# B&R Automation Studio project NAEUL004C00R13L518F00 (part 23)

#### Act_OptP0939FBCtrl.st
```iecst
ACTION Act_OptP0939FBCtrl:

	fbJogSlowToFastDlyTm.PT	:= T#2s;
	fbJogSlowToFastDlyTm;
	fbLmtRstTm;

	//Lifter Safety Sensor Interruption
	IF EDGENEG(p_tyDI.bLifterSafetyLmtSW1 AND p_tyDI.bLifterSafetyLmtSW2 AND p_tyDI.bLifterTimingBeltSen) THEN
		tyP0939Lifter2.tyMotionStd.tyBtnStop.bRtCompl	:= TRUE;
	END_IF

//	IF EDGEPOS((p_udiLifter2AxisErrID = 21570 OR p_udiLifter2AxisErrID = 21571)
	IF EDGEPOS((p_bLifter2FwdLmtSen OR p_bLifter2RevLmtSen OR p_udiLifter2AxisErrID = 21570 OR p_udiLifter2AxisErrID = 21571)
		AND tyP0939Lifter2.tyMotionStd.tyBtnJogDown.bValue = FALSE
		AND tyP0939Lifter2.tyMotionStd.tyBtnJogUp.bValue = FALSE)
	THEN
		fbLmtRstTm.IN				:= TRUE;
	END_IF

	IF fbLmtRstTm.Q = TRUE THEN
		tyP0939Lifter2.tyMotionStd.tyBtnRst.bRtCompl		:= TRUE;
	END_IF

	IF (tyP0939Lifter2.tyMotionStd.tyBtnJogUp.bValue = FALSE AND tyP0939Lifter2.tyMotionStd.tyBtnJogDown.bValue = FALSE) AND (p_bLifter2Jogging = TRUE) THEN
		bJogStopLifter	:= TRUE;
	END_IF

	IF tyP0939Lifter2.tyMotionStd.tyBtnStop.bRtCompl = TRUE THEN
		eLifter2Act		:= LifterActStop;

		IF p_eLifter2Stat = LifterActStop AND p_eLifter2Status = Done THEN
			eLifter2Act	:= LifterActIdle;

			tyP0939Lifter2.tyMotionStd.tyBtnStop.bRtCompl			:= FALSE;
			tyP0939Lifter2.tyMotionStd.tyBtnJogDown.bRtCompl			:= FALSE;
			tyP0939Lifter2.tyMotionStd.tyBtnJogUp.bRtCompl			:= FALSE;
			tyP0939Lifter2.tyMotionStd.tyBtnOrigin.bRtCompl			:= FALSE;
			tyP0939Lifter2.tyMotionStd.tyBtnMovAbs.bRtCompl			:= FALSE;
			tyP0939Lifter2.tyMotionStd.tyBtnMovRel.bRtCompl			:= FALSE;
			tyP0939Lifter2.tyLifter.tyBtnGo.bRtCompl				:= FALSE;
			tyP0939Lifter2.tyLifter.tyBtnNxtSlt.bRtCompl			:= FALSE;
			tyP0939Lifter2.tyLifter.tyBtnPrevSlt.bRtCompl			:= FALSE;
			tyP0939Lifter2.tyLifter.tyBtnGoLaneA.bRtCompl			:= FALSE;
			tyP0939Lifter2.tyLifter.tyBtnGoLaneB.bRtCompl			:= FALSE;
			tyP0939Lifter2.tyLifter.tyBtnGoLaneD_G.bRtCompl			:= FALSE;
			tyP0939Lifter2.tyLifter.tyBtnGoLaneE_H.bRtCompl			:= FALSE;

			tyP0939Lifter2.tyMotionStd.tyBtnStop.bValue				:= TRUE;
			tyP0939Lifter2.tyMotionStd.tyBtnJogDown.bValue			:= FALSE;
			tyP0939Lifter2.tyMotionStd.tyBtnJogUp.bValue				:= FALSE;
			tyP0939Lifter2.tyMotionStd.tyBtnOrigin.bValue			:= FALSE;
			tyP0939Lifter2.tyMotionStd.tyBtnMovAbs.bValue			:= FALSE;
			tyP0939Lifter2.tyMotionStd.tyBtnMovRel.bValue			:= FALSE;
			tyP0939Lifter2.tyLifter.tyBtnGo.bValue					:= FALSE;
			tyP0939Lifter2.tyLifter.tyBtnNxtSlt.bValue				:= FALSE;
			tyP0939Lifter2.tyLifter.tyBtnPrevSlt.bValue				:= FALSE;
			tyP0939Lifter2.tyLifter.tyBtnGoLaneA.bValue				:= FALSE;
			tyP0939Lifter2.tyLifter.tyBtnGoLaneB.bValue				:= FALSE;
			tyP0939Lifter2.tyLifter.tyBtnGoLaneD_G.bValue			:= FALSE;
			tyP0939Lifter2.tyLifter.tyBtnGoLaneE_H.bValue			:= FALSE;

			tyP0939Lifter2.tyMotionStd.tyBtnStop.bRtLk				:= TRUE;
			tyP0939Lifter2.tyMotionStd.tyBtnJogDown.bRtLk			:= FALSE;
			tyP0939Lifter2.tyMotionStd.tyBtnJogUp.bRtLk				:= FALSE;
			tyP0939Lifter2.tyMotionStd.tyBtnOrigin.bRtLk				:= FALSE;
			tyP0939Lifter2.tyMotionStd.tyBtnMovAbs.bRtLk				:= FALSE;
			tyP0939Lifter2.tyMotionStd.tyBtnMovRel.bRtLk				:= FALSE;
			tyP0939Lifter2.tyLifter.tyBtnGo.bRtLk					:= FALSE;
			tyP0939Lifter2.tyLifter.tyBtnNxtSlt.bRtLk				:= FALSE;
			tyP0939Lifter2.tyLifter.tyBtnPrevSlt.bRtLk				:= FALSE;
			tyP0939Lifter2.tyLifter.tyBtnGoLaneA.bRtLk				:= FALSE;
			tyP0939Lifter2.tyLifter.tyBtnGoLaneB.bRtLk				:= FALSE;
			tyP0939Lifter2.tyLifter.tyBtnGoLaneD_G.bRtLk			:= FALSE;
			tyP0939Lifter2.tyLifter.tyBtnGoLaneE_H.bRtLk			:= FALSE;

		END_IF

	ELSIF (tyP0939Lifter2.tyMotionStd.tyBtnJogDown.bRtCompl = TRUE) OR (tyP0939Lifter2.tyMotionStd.tyBtnJogUp.bRtCompl = TRUE) OR (bJogStopLifter = TRUE) THEN
		bJogSlow					:= FALSE;
		bJogFast					:= FALSE;
		fbJogSlowToFastDlyTm.IN		:= FALSE;

		eLifter2Act		:= LifterActJogStop;

		IF p_eLifter2Stat = LifterActJogStop AND p_eLifter2Status = Done THEN
			eLifter2Act		:= LifterActIdle;

			bJogStopLifter	:= FALSE;

			tyP0939Lifter2.tyMotionStd.tyBtnStop.bRtCompl			:= FALSE;
			tyP0939Lifter2.tyMotionStd.tyBtnJogDown.bRtCompl		:= FALSE;
			tyP0939Lifter2.tyMotionStd.tyBtnJogUp.bRtCompl			:= FALSE;
			tyP0939Lifter2.tyMotionStd.tyBtnOrigin.bRtCompl			:= FALSE;
			tyP0939Lifter2.tyMotionStd.tyBtnMovAbs.bRtCompl			:= FALSE;
			tyP0939Lifter2.tyMotionStd.tyBtnMovRel.bRtCompl			:= FALSE;
			tyP0939Lifter2.tyLifter.tyBtnGo.bRtCompl				:= FALSE;
			tyP0939Lifter2.tyLifter.tyBtnNxtSlt.bRtCompl			:= FALSE;
			tyP0939Lifter2.tyLifter.tyBtnPrevSlt.bRtCompl			:= FALSE;
			tyP0939Lifter2.tyLifter.tyBtnGoLaneA.bRtCompl			:= FALSE;
			tyP0939Lifter2.tyLifter.tyBtnGoLaneB.bRtCompl			:= FALSE;
			tyP0939Lifter2.tyLifter.tyBtnGoLaneD_G.bRtCompl			:= FALSE;
			tyP0939Lifter2.tyLifter.tyBtnGoLaneE_H.bRtCompl			:= FALSE;

			tyP0939Lifter2.tyMotionStd.tyBtnStop.bValue				:= TRUE;
			tyP0939Lifter2.tyMotionStd.tyBtnJogDown.bValue			:= FALSE;
			tyP0939Lifter2.tyMotionStd.tyBtnJogUp.bValue			:= FALSE;
			tyP0939Lifter2.tyMotionStd.tyBtnOrigin.bValue			:= FALSE;
			tyP0939Lifter2.tyMotionStd.tyBtnMovAbs.bValue			:= FALSE;
			tyP0939Lifter2.tyMotionStd.tyBtnMovRel.bValue			:= FALSE;
			tyP0939Lifter2.tyLifter.tyBtnGo.bValue					:= FALSE;
			tyP0939Lifter2.tyLifter.tyBtnNxtSlt.bValue				:= FALSE;
			tyP0939Lifter2.tyLifter.tyBtnPrevSlt.bValue				:= FALSE;
			tyP0939Lifter2.tyLifter.tyBtnGoLaneA.bValue				:= FALSE;
			tyP0939Lifter2.tyLifter.tyBtnGoLaneB.bValue				:= FALSE;
			tyP0939Lifter2.tyLifter.tyBtnGoLaneD_G.bValue			:= FALSE;
			tyP0939Lifter2.tyLifter.tyBtnGoLaneE_H.bValue			:= FALSE;

			tyP0939Lifter2.tyMotionStd.tyBtnStop.bRtLk				:= TRUE;
			tyP0939Lifter2.tyMotionStd.tyBtnJogDown.bRtLk			:= FALSE;
			tyP0939Lifter2.tyMotionStd.tyBtnJogUp.bRtLk				:= FALSE;
			tyP0939Lifter2.tyMotionStd.tyBtnOrigin.bRtLk			:= FALSE;
			tyP0939Lifter2.tyMotionStd.tyBtnMovAbs.bRtLk			:= FALSE;
			tyP0939Lifter2.tyMotionStd.tyBtnMovRel.bRtLk			:= FALSE;
			tyP0939Lifter2.tyLifter.tyBtnGo.bRtLk					:= FALSE;
			tyP0939Lifter2.tyLifter.tyBtnNxtSlt.bRtLk				:= FALSE;
			tyP0939Lifter2.tyLifter.tyBtnPrevSlt.bRtLk				:= FALSE;
			tyP0939Lifter2.tyLifter.tyBtnGoLaneA.bRtLk				:= FALSE;
			tyP0939Lifter2.tyLifter.tyBtnGoLaneB.bRtLk				:= FALSE;
			tyP0939Lifter2.tyLifter.tyBtnGoLaneD_G.bRtLk			:= FALSE;
			tyP0939Lifter2.tyLifter.tyBtnGoLaneE_H.bRtLk			:= FALSE;

		END_IF

	ELSIF tyP0939Lifter2.tyMotionStd.tyBtnPwr.bRtCompl = TRUE THEN
		tyP0939Lifter2.tyMotionStd.tyBtnPwr.bRtLk					:= TRUE;

		IF tyP0939Lifter2.tyMotionStd.tyBtnPwr.bValue = TRUE THEN
			eLifter2Act		:= LifterActPwrOn;

			IF p_eLifter2Stat = LifterActPwrOn AND p_eLifter2Status = Done THEN
				eLifter2Act	:= LifterActIdle;

				tyP0939Lifter2.tyMotionStd.tyBtnPwr.bRtCompl		:= FALSE;
				tyP0939Lifter2.tyMotionStd.tyBtnPwr.bRtLk		:= FALSE;
			END_IF
		ELSE
			eLifter2Act		:= LifterActPwrOff;

			IF p_eLifter2Stat = LifterActPwrOff AND p_eLifter2Status = Done THEN
				eLifter2Act	:= LifterActIdle;

				tyP0939Lifter2.tyMotionStd.tyBtnPwr.bRtCompl		:= FALSE;
				tyP0939Lifter2.tyMotionStd.tyBtnPwr.bRtLk		:= FALSE;
			END_IF
		END_IF

	ELSIF tyP0939Lifter2.tyMotionStd.tyBtnOrigin.bRtCompl = TRUE THEN
		tyP0939Lifter2.tyMotionStd.tyBtnOrigin.bValue				:= TRUE;
		tyP0939Lifter2.tyMotionStd.tyBtnStop.bValue					:= FALSE;

		tyP0939Lifter2.tyMotionStd.tyBtnOrigin.bRtLk					:= TRUE;
		tyP0939Lifter2.tyMotionStd.tyBtnStop.bRtLk					:= FALSE;

		eLifter2Act		:= LifterActHoming;

		IF p_eLifter2Stat = LifterActHoming AND p_eLifter2Status = Done THEN
			eLifter2Act	:= LifterActIdle;

			tyP0939Lifter2.tyMotionStd.tyBtnOrigin.bRtCompl		:= FALSE;
			tyP0939Lifter2.tyMotionStd.tyBtnOrigin.bValue		:= FALSE;
			tyP0939Lifter2.tyMotionStd.tyBtnStop.bValue			:= TRUE;

			tyP0939Lifter2.tyMotionStd.tyBtnOrigin.bRtLk			:= FALSE;
			tyP0939Lifter2.tyMotionStd.tyBtnStop.bRtLk			:= TRUE;

		END_IF

	ELSIF tyP0939Lifter2.tyMotionStd.tyBtnRst.bRtCompl = TRUE THEN
		tyP0939Lifter2.tyMotionStd.tyBtnRst.bValue				:= TRUE;
		tyP0939Lifter2.tyMotionStd.tyBtnRst.bRtLk				:= TRUE;

		eLifter2Act		:= LifterActRstAxisErr;

		IF p_eLifter2Stat = LifterActRstAxisErr AND p_eLifter2Status = Done THEN
			eLifter2Act	:= LifterActIdle;

			tyP0939Lifter2.tyMotionStd.tyBtnRst.bRtCompl			:= FALSE;
			tyP0939Lifter2.tyMotionStd.tyBtnRst.bValue			:= FALSE;
			tyP0939Lifter2.tyMotionStd.tyBtnRst.bRtLk			:= FALSE;

			fbLmtRstTm.IN			:= FALSE;
		END_IF

	ELSIF tyP0939Lifter2.tyLifter.tyBtnGo.bRtCompl = TRUE THEN
		tyP0939Lifter2.tyLifter.tyBtnGo.bValue				:= TRUE;
		tyP0939Lifter2.tyMotionStd.tyBtnStop.bValue			:= FALSE;

		tyP0939Lifter2.tyLifter.tyBtnGo.bRtLk				:= TRUE;
		tyP0939Lifter2.tyMotionStd.tyBtnStop.bRtLk			:= FALSE;

		(*diMnlLifterMag1GoSlt2	:= tyP0939Lifter2.tyLifter.tyNumNewSlt.diValue;*)
		diMnlLifterNomSpd2		:= tyP0939Lifter2.tyMotionStd.tyNumNomSpd.diValue;

		CASE tyP0939Lifter2.tyLifter.tyNumMagPos.diValue OF
			1:
				eLifter2Act	:= LifterActGoASltPos;
				diMnlLifterMag1GoSlt2	:= tyP0939Lifter2.tyLifter.tyNumNewSlt.diValue;

			2:
				eLifter2Act	:= LifterActGoBSltPos;
				diMnlLifterMag2GoSlt2	:= tyP0939Lifter2.tyLifter.tyNumNewSlt.diValue;

			3:
				eLifter2Act	:= LifterActGoCSltPos;
				diMnlLifterMag3GoSlt2	:= tyP0939Lifter2.tyLifter.tyNumNewSlt.diValue;

			4:
				eLifter2Act	:= LifterActGoDSltPos;
				diMnlLifterMag3GoSlt2	:= tyP0939Lifter2.tyLifter.tyNumNewSlt.diValue;
		END_CASE

		IF (p_eLifter2Stat = LifterActGoASltPos
			OR p_eLifter2Stat = LifterActGoBSltPos
			OR p_eLifter2Stat = LifterActGoCSltPos
			OR p_eLifter2Stat = LifterActGoDSltPos)
			AND p_eLifter2Status = Done THEN
			eLifter2Act	:= LifterActIdle;

			tyP0939Lifter2.tyLifter.tyBtnGo.bRtCompl				:= FALSE;
			tyP0939Lifter2.tyLifter.tyBtnGo.bValue				:= FALSE;
			tyP0939Lifter2.tyMotionStd.tyBtnStop.bValue			:= TRUE;

			tyP0939Lifter2.tyLifter.tyBtnGo.bRtLk				:= FALSE;
			tyP0939Lifter2.tyMotionStd.tyBtnStop.bRtLk			:= TRUE;
		END_IF

	ELSIF tyP0939Lifter2.tyLifter.tyBtnNxtSlt.bRtCompl = TRUE THEN
		tyP0939Lifter2.tyLifter.tyBtnNxtSlt.bValue				:= TRUE;
		tyP0939Lifter2.tyMotionStd.tyBtnStop.bValue				:= FALSE;

		tyP0939Lifter2.tyLifter.tyBtnNxtSlt.bRtLk				:= TRUE;
		tyP0939Lifter2.tyMotionStd.tyBtnStop.bRtLk				:= FALSE;

		(*diMnlLifterMag1GoSlt2	:= tyP0939Lifter2.tyLifter.tyNumNewSlt.diValue;*)
		diMnlLifterNomSpd2		:= tyP0939Lifter2.tyMotionStd.tyNumNomSpd.diValue;

		CASE tyP0939Lifter2.tyLifter.tyNumMagPos.diValue OF
			1:
				eLifter2Act	:= LifterActGoNxtASltPos;
				diMnlLifterMag1GoSlt2	:= tyP0939Lifter2.tyLifter.tyNumNewSlt.diValue;
			2:
				eLifter2Act	:= LifterActGoNxtBSltPos;
				diMnlLifterMag2GoSlt2	:= tyP0939Lifter2.tyLifter.tyNumNewSlt.diValue;
			3:
				eLifter2Act	:= LifterActGoNxtCSltPos;
				diMnlLifterMag3GoSlt2	:= tyP0939Lifter2.tyLifter.tyNumNewSlt.diValue;
			4:
				eLifter2Act	:= LifterActGoNxtDSltPos;
		//		diMnlLifterMag4GoSlt	:= tyP0939Lifter2.tyLifter.tyNumNewSlt.diValue;

		END_CASE

		IF (p_eLifter2Stat = LifterActGoNxtASltPos
			OR p_eLifter2Stat = LifterActGoNxtBSltPos
			OR p_eLifter2Stat = LifterActGoNxtCSltPos
			OR p_eLifter2Stat = LifterActGoNxtDSltPos)
			AND p_eLifter2Status = Done THEN
			eLifter2Act	:= LifterActIdle;

			tyP0939Lifter2.tyLifter.tyBtnNxtSlt.bRtCompl				:= FALSE;
			tyP0939Lifter2.tyLifter.tyBtnNxtSlt.bValue				:= FALSE;
			tyP0939Lifter2.tyMotionStd.tyBtnStop.bValue				:= TRUE;

			tyP0939Lifter2.tyLifter.tyBtnNxtSlt.bRtLk				:= FALSE;
			tyP0939Lifter2.tyMotionStd.tyBtnStop.bRtLk				:= TRUE;
		END_IF

	ELSIF tyP0939Lifter2.tyLifter.tyBtnPrevSlt.bRtCompl = TRUE THEN
		tyP0939Lifter2.tyLifter.tyBtnPrevSlt.bValue				:= TRUE;
		tyP0939Lifter2.tyMotionStd.tyBtnStop.bValue				:= FALSE;

		tyP0939Lifter2.tyLifter.tyBtnPrevSlt.bRtLk				:= TRUE;
		tyP0939Lifter2.tyMotionStd.tyBtnStop.bRtLk				:= FALSE;

	//	diMnlLifterMag1GoSlt2	:= tyP0939Lifter2.tyLifter.tyNumNewSlt.diValue;
		diMnlLifterNomSpd2		:= tyP0939Lifter2.tyMotionStd.tyNumNomSpd.diValue;

		CASE tyP0939Lifter2.tyLifter.tyNumMagPos.diValue OF

			1:
				eLifter2Act	:= LifterActGoPrevASltPos;
				diMnlLifterMag1GoSlt2	:= tyP0939Lifter2.tyLifter.tyNumNewSlt.diValue;

			2:
				eLifter2Act	:= LifterActGoPrevBSltPos;
				diMnlLifterMag2GoSlt2	:= tyP0939Lifter2.tyLifter.tyNumNewSlt.diValue;

			3:
				eLifter2Act	:= LifterActGoPrevCSltPos;
				diMnlLifterMag3GoSlt2	:= tyP0939Lifter2.tyLifter.tyNumNewSlt.diValue;

			4:
				eLifter2Act	:= LifterActGoPrevDSltPos;
		//		diMnlLifterMag4GoSlt	:= tyP0939Lifter2.tyLifter.tyNumNewSlt.diValue;

		END_CASE

		IF (p_eLifter2Stat = LifterActGoPrevASltPos
			OR p_eLifter2Stat = LifterActGoPrevBSltPos
			OR p_eLifter2Stat = LifterActGoPrevCSltPos
			OR p_eLifter2Stat = LifterActGoPrevDSltPos)
			AND p_eLifter2Status = Done THEN
			eLifter2Act	:= LifterActIdle;

			tyP0939Lifter2.tyLifter.tyBtnPrevSlt.bRtCompl				:= FALSE;
			tyP0939Lifter2.tyLifter.tyBtnPrevSlt.bValue					:= FALSE;
			tyP0939Lifter2.tyMotionStd.tyBtnStop.bValue					:= TRUE;

			tyP0939Lifter2.tyLifter.tyBtnPrevSlt.bRtLk					:= FALSE;
			tyP0939Lifter2.tyMotionStd.tyBtnStop.bRtLk					:= TRUE;
		END_IF

	ELSIF tyP0939Lifter2.tyLifter.tyBtnGoLaneA.bRtCompl = TRUE THEN
		tyP0939Lifter2.tyLifter.tyBtnGoLaneA.bValue	:= TRUE;
		tyP0939Lifter2.tyMotionStd.tyBtnStop.bValue	:= FALSE;

		tyP0939Lifter2.tyLifter.tyBtnGoLaneA.bRtLk	:= TRUE;
		tyP0939Lifter2.tyMotionStd.tyBtnStop.bRtLk	:= FALSE;

		diMnlLifterNomSpd2	:= tyP0939Lifter2.tyMotionStd.tyNumNomSpd.diValue;

		eLifter2Act	:= LifterActGoAPos;

		IF p_eLifter2Stat = LifterActGoAPos AND p_eLifter2Status = Done THEN
			eLifter2Act	:= LifterActIdle;

			tyP0939Lifter2.tyLifter.tyBtnGoLaneA.bRtCompl	:= FALSE;

			tyP0939Lifter2.tyLifter.tyBtnGoLaneA.bValue	:= FALSE;
			tyP0939Lifter2.tyMotionStd.tyBtnStop.bValue	:= TRUE;

			tyP0939Lifter2.tyLifter.tyBtnGoLaneA.bRtLk	:= FALSE;
			tyP0939Lifter2.tyMotionStd.tyBtnStop.bRtLk	:= TRUE;
		END_IF

	ELSIF tyP0939Lifter2.tyLifter.tyBtnGoLaneB.bRtCompl = TRUE THEN
		tyP0939Lifter2.tyLifter.tyBtnGoLaneB.bValue	:= TRUE;
		tyP0939Lifter2.tyMotionStd.tyBtnStop.bValue	:= FALSE;

		tyP0939Lifter2.tyLifter.tyBtnGoLaneB.bRtLk	:= TRUE;
		tyP0939Lifter2.tyMotionStd.tyBtnStop.bRtLk	:= FALSE;

		diMnlLifterNomSpd2	:= tyP0939Lifter2.tyMotionStd.tyNumNomSpd.diValue;

		eLifter2Act	:= LifterActGoBPos;

		IF p_eLifter2Stat = LifterActGoBPos AND p_eLifter2Status = Done THEN
			eLifter2Act	:= LifterActIdle;

			tyP0939Lifter2.tyLifter.tyBtnGoLaneB.bRtCompl	:= FALSE;

			tyP0939Lifter2.tyLifter.tyBtnGoLaneB.bValue	:= FALSE;
			tyP0939Lifter2.tyMotionStd.tyBtnStop.bValue	:= TRUE;

			tyP0939Lifter2.tyLifter.tyBtnGoLaneB.bRtLk	:= FALSE;
			tyP0939Lifter2.tyMotionStd.tyBtnStop.bRtLk	:= TRUE;
		END_IF

	ELSIF tyP0939Lifter2.tyLifter.tyBtnGoLaneD_G.bRtCompl = TRUE THEN
		tyP0939Lifter2.tyLifter.tyBtnGoLaneD_G.bValue	:= TRUE;
		tyP0939Lifter2.tyMotionStd.tyBtnStop.bValue	:= FALSE;

		tyP0939Lifter2.tyLifter.tyBtnGoLaneD_G.bRtLk	:= TRUE;
		tyP0939Lifter2.tyMotionStd.tyBtnStop.bRtLk	:= FALSE;

		diMnlLifterNomSpd2	:= tyP0939Lifter2.tyMotionStd.tyNumNomSpd.diValue;

		eLifter2Act	:= LifterActGoGPos;

		IF p_eLifter2Stat = LifterActGoGPos AND p_eLifter2Status = Done THEN
			eLifter2Act	:= LifterActIdle;

			tyP0939Lifter2.tyLifter.tyBtnGoLaneD_G.bRtCompl	:= FALSE;

			tyP0939Lifter2.tyLifter.tyBtnGoLaneD_G.bValue	:= FALSE;
			tyP0939Lifter2.tyMotionStd.tyBtnStop.bValue	:= TRUE;

			tyP0939Lifter2.tyLifter.tyBtnGoLaneD_G.bRtLk	:= FALSE;
			tyP0939Lifter2.tyMotionStd.tyBtnStop.bRtLk	:= TRUE;
		END_IF

	ELSIF tyP0939Lifter2.tyLifter.tyBtnGoLaneE_H.bRtCompl = TRUE THEN
		tyP0939Lifter2.tyLifter.tyBtnGoLaneE_H.bValue	:= TRUE;
		tyP0939Lifter2.tyMotionStd.tyBtnStop.bValue	:= FALSE;

		tyP0939Lifter2.tyLifter.tyBtnGoLaneE_H.bRtLk	:= TRUE;
		tyP0939Lifter2.tyMotionStd.tyBtnStop.bRtLk	:= FALSE;

		diMnlLifterNomSpd2	:= tyP0939Lifter2.tyMotionStd.tyNumNomSpd.diValue;

		eLifter2Act	:= LifterActGoHPos;

		IF p_eLifter2Stat = LifterActGoHPos AND p_eLifter2Status = Done THEN
			eLifter2Act	:= LifterActIdle;

			tyP0939Lifter2.tyLifter.tyBtnGoLaneE_H.bRtCompl	:= FALSE;

			tyP0939Lifter2.tyLifter.tyBtnGoLaneE_H.bValue	:= FALSE;
			tyP0939Lifter2.tyMotionStd.tyBtnStop.bValue	:= TRUE;

			tyP0939Lifter2.tyLifter.tyBtnGoLaneE_H.bRtLk	:= FALSE;
			tyP0939Lifter2.tyMotionStd.tyBtnStop.bRtLk	:= TRUE;
		END_IF
	ELSIF tyP0939Lifter2.tyMotionStd.tyBtnMovAbs.bRtCompl = TRUE THEN

		tyP0939Lifter2.tyMotionStd.tyBtnMovAbs.bValue				:= TRUE;
		tyP0939Lifter2.tyMotionStd.tyBtnStop.bValue					:= FALSE;

		tyP0939Lifter2.tyMotionStd.tyBtnMovAbs.bRtLk					:= TRUE;
		tyP0939Lifter2.tyMotionStd.tyBtnStop.bRtLk					:= FALSE;

		diMnlLifterTargetPos2	:= tyP0939Lifter2.tyMotionStd.tyNumTargetPos.diValue;
		diMnlLifterNomSpd2		:= tyP0939Lifter2.tyMotionStd.tyNumNomSpd.diValue;

		eLifter2Act			:= LifterActMovAbs;

		IF p_eLifter2Stat = LifterActMovAbs AND p_eLifter2Status = Done THEN
			eLifter2Act	:= LifterActIdle;

			tyP0939Lifter2.tyMotionStd.tyBtnMovAbs.bRtCompl		:= FALSE;
			tyP0939Lifter2.tyMotionStd.tyBtnMovAbs.bValue		:= FALSE;
			tyP0939Lifter2.tyMotionStd.tyBtnStop.bValue			:= TRUE;

			tyP0939Lifter2.tyMotionStd.tyBtnMovAbs.bRtLk			:= FALSE;
			tyP0939Lifter2.tyMotionStd.tyBtnStop.bRtLk			:= TRUE;
		END_IF

	ELSIF tyP0939Lifter2.tyMotionStd.tyBtnMovRel.bRtCompl = TRUE THEN
		tyP0939Lifter2.tyMotionStd.tyBtnMovRel.bValue			:= TRUE;
		tyP0939Lifter2.tyMotionStd.tyBtnStop.bValue				:= FALSE;

		tyP0939Lifter2.tyMotionStd.tyBtnMovRel.bRtLk				:= TRUE;
		tyP0939Lifter2.tyMotionStd.tyBtnStop.bRtLk				:= FALSE;

		diMnlLifterStepSize2		:= tyP0939Lifter2.tyMotionStd.tyNumStepSize.diValue;
		diMnlLifterNomSpd2		:= tyP0939Lifter2.tyMotionStd.tyNumNomSpd.diValue;

		eLifter2Act		:= LifterActMovRel;

		IF p_eLifter2Stat = LifterActMovRel AND p_eLifter2Status = Done THEN
			eLifter2Act	:= LifterActIdle;

			tyP0939Lifter2.tyMotionStd.tyBtnMovRel.bRtCompl		:= FALSE;
			tyP0939Lifter2.tyMotionStd.tyBtnMovRel.bValue		:= FALSE;
			tyP0939Lifter2.tyMotionStd.tyBtnStop.bValue			:= TRUE;

			tyP0939Lifter2.tyMotionStd.tyBtnMovRel.bRtLk			:= FALSE;
			tyP0939Lifter2.tyMotionStd.tyBtnStop.bRtLk			:= TRUE;

		END_IF

	ELSIF (tyP0939Lifter2.tyMotionStd.tyBtnJogDown.bValue = TRUE) AND (fbJogSlowToFastDlyTm.Q = FALSE) AND (bJogSlow = FALSE) THEN
		tyP0939Lifter2.tyMotionStd.tyBtnStop.bValue				:= FALSE;
		tyP0939Lifter2.tyMotionStd.tyBtnStop.bRtLk				:= FALSE;

		fbJogSlowToFastDlyTm.IN		:= TRUE;

		diMnlLifterJogSpd2	:= tyP0939Lifter2.tyMotionStd.tyNumSlwSpd.diValue;

		eLifter2Act		:= LifterActJogDown;

		IF p_eLifter2Stat = LifterActJogDown AND p_eLifter2Status = Done THEN

			eLifter2Act	:= LifterActIdle;
			bJogSlow				:= TRUE;

		ELSIF p_eLifter2Status = Error THEN

			fbJogSlowToFastDlyTm.IN	:= FALSE;
			bJogSlow				:= TRUE;

		END_IF

	ELSIF (tyP0939Lifter2.tyMotionStd.tyBtnJogDown.bValue = TRUE) AND (fbJogSlowToFastDlyTm.Q = TRUE) AND (bJogFast = FALSE) THEN
		tyP0939Lifter2.tyMotionStd.tyBtnStop.bValue					:= FALSE;
		tyP0939Lifter2.tyMotionStd.tyBtnStop.bRtLk					:= FALSE;

		fbJogSlowToFastDlyTm.IN		:= TRUE;

		diMnlLifterJogSpd2	:= tyP0939Lifter2.tyMotionStd.tyNumNomSpd.diValue;

		eLifter2Act		:= LifterActJogDown;

		IF p_eLifter2Stat = LifterActJogDown AND p_eLifter2Status = Done THEN
			eLifter2Act	:= LifterActIdle;
			bJogFast				:= TRUE;
		ELSIF p_eLifter2Status = Error THEN
			fbJogSlowToFastDlyTm.IN	:= FALSE;
			bJogFast				:= TRUE;
		END_IF

	ELSIF (tyP0939Lifter2.tyMotionStd.tyBtnJogUp.bValue = TRUE) AND (fbJogSlowToFastDlyTm.Q = FALSE) AND (bJogSlow = FALSE) THEN
		tyP0939Lifter2.tyMotionStd.tyBtnStop.bValue				:= FALSE;
		tyP0939Lifter2.tyMotionStd.tyBtnStop.bRtLk				:= FALSE;

		fbJogSlowToFastDlyTm.IN		:= TRUE;

		diMnlLifterJogSpd2	:= tyP0939Lifter2.tyMotionStd.tyNumSlwSpd.diValue;

		eLifter2Act		:= LifterActJogUp;

		IF p_eLifter2Stat = LifterActJogUp AND p_eLifter2Status = Done THEN
			eLifter2Act	:= LifterActIdle;
			bJogSlow				:= TRUE;

		ELSIF p_eLifter2Status = Error THEN
			fbJogSlowToFastDlyTm.IN	:= FALSE;
			bJogSlow				:= TRUE;
		END_IF

	ELSIF (tyP0939Lifter2.tyMotionStd.tyBtnJogUp.bValue = TRUE) AND (fbJogSlowToFastDlyTm.Q = TRUE) AND (bJogFast = FALSE) THEN

		tyP0939Lifter2.tyMotionStd.tyBtnStop.bValue				:= FALSE;
		tyP0939Lifter2.tyMotionStd.tyBtnStop.bRtLk				:= FALSE;

		fbJogSlowToFastDlyTm.IN		:= TRUE;

		diMnlLifterJogSpd2	:= tyP0939Lifter2.tyMotionStd.tyNumNomSpd.diValue;

		eLifter2Act		:= LifterActJogUp;

		IF p_eLifter2Stat = LifterActJogUp AND p_eLifter2Status = Done THEN
			eLifter2Act	:= LifterActIdle;
			bJogFast	:= TRUE;

		ELSIF p_eLifter2Status = Error THEN
			fbJogSlowToFastDlyTm.IN	:= FALSE;
			bJogFast				:= TRUE;
		END_IF
	END_IF

	//Shutter Control
	IF tyP0939Lifter2.tyInOutletShutterFB.tyBtnOpen.bRtCompl = TRUE THEN
		tyP0939Lifter2.tyInOutletShutterFB.tyBtnOpen.bRtCompl	:= FALSE;

		tyP0939Lifter2.tyInOutletShutterFB.tyBtnOpen.bValue	:= TRUE;
		tyP0939Lifter2.tyInOutletShutterFB.tyBtnClose.bValue	:= FALSE;

	ELSIF tyP0939Lifter2.tyInOutletShutterFB.tyBtnClose.bRtCompl = TRUE THEN
		tyP0939Lifter2.tyInOutletShutterFB.tyBtnClose.bRtCompl	:= FALSE;

		tyP0939Lifter2.tyInOutletShutterFB.tyBtnClose.bValue	:= TRUE;
		tyP0939Lifter2.tyInOutletShutterFB.tyBtnOpen.bValue	:= FALSE;
	END_IF

	IF tyP0939Lifter2.tyInOutletShutterFB.tyBtnOpen.bValue = TRUE THEN
		eInShutterAct	:= PneuActRet;
		eOutShutterAct	:= PneuActRet;

		IF (p_eInShutterStat = PneuActRet AND p_eInShutterStatus = Done)
			AND (p_eOutShutterStat = PneuActRet AND p_eOutShutterStatus = Done)
			THEN
			eInShutterAct	:= PneuActIdle;
			eOutShutterAct	:= PneuActIdle;
			tyP0939Lifter2.tyInOutletShutterFB.tyBtnOpen.bValue	:= FALSE;
		ELSIF p_eInShutterStatus = Error OR p_eOutShutterStatus = Error THEN
			tyP0939Lifter2.tyInOutletShutterFB.tyBtnOpen.bValue	:= FALSE;
		END_IF

	ELSIF tyP0939Lifter2.tyInOutletShutterFB.tyBtnClose.bValue = TRUE THEN
		eInShutterAct	:= PneuActExt;
		eOutShutterAct	:= PneuActExt;
		IF (p_eInShutterStat = PneuActExt AND p_eInShutterStatus = Done)
			AND (p_eOutShutterStat = PneuActExt AND p_eOutShutterStatus = Done)
			THEN
			eInShutterAct	:= PneuActIdle;
			eOutShutterAct	:= PneuActIdle;
			tyP0939Lifter2.tyInOutletShutterFB.tyBtnClose.bValue := FALSE;
		ELSIF p_eInShutterStatus = Error OR p_eOutShutterStatus = Error THEN
			tyP0939Lifter2.tyInOutletShutterFB.tyBtnClose.bValue := FALSE;
		END_IF
	END_IF

END_ACTION
```

#### Act_OptP0939FBStat.st
```iecst
ACTION Act_OptP0939FBStat:

	IF p_bLifter2AxisErr = TRUE THEN
		tyP0939Lifter2.tyMotionStd.tyStringStat.sValue	:= p_sLifter2AxisErrTxt;
	ELSE
		IF NOT(p_bLifter2Jogging AND p_eLifter2Stat = LifterActIdle) THEN
			tyP0939Lifter2.tyMotionStd.tyStringStat.sValue	:= p_sLifter2StatTxt;
		END_IF
	END_IF

END_ACTION
```

#### Act_OptP0939Mask.st
```iecst
ACTION Act_OptP0939Mask:

	// Interlock Power
	IF p_bLifter2AxisErr = TRUE AND p_bLifter2PwrOn = FALSE THEN
		fUIInRtStatOff(ADR(tyP0939Lifter2.tyMotionStd.tyBtnPwr.uiMaskRtStat));
		tyP0939Lifter2.tyMotionStd.tyBtnPwr.bValue		:= FALSE;
	ELSE
		fUIInRtStatHide(ADR(tyP0939Lifter2.tyMotionStd.tyBtnPwr.uiMaskRtStat));
	END_IF

	// Interlock Others Move
	IF p_bLifter2AxisErr = TRUE OR p_bLifter2PwrOn = FALSE THEN
		fUIInRtStatOff(ADR(tyP0939Lifter2.tyMotionStd.tyBtnOrigin.uiMaskRtStat));
		fUIInRtStatOff(ADR(tyP0939Lifter2.tyMotionStd.tyBtnMovRel.uiMaskRtStat));
		fUIInRtStatOff(ADR(tyP0939Lifter2.tyMotionStd.tyBtnJogUp.uiMaskRtStat));
		fUIInRtStatOff(ADR(tyP0939Lifter2.tyMotionStd.tyBtnJogDown.uiMaskRtStat));
	ELSE
		fUIInRtStatHide(ADR(tyP0939Lifter2.tyMotionStd.tyBtnOrigin.uiMaskRtStat));
		fUIInRtStatHide(ADR(tyP0939Lifter2.tyMotionStd.tyBtnMovRel.uiMaskRtStat));
		fUIInRtStatHide(ADR(tyP0939Lifter2.tyMotionStd.tyBtnJogUp.uiMaskRtStat));
		fUIInRtStatHide(ADR(tyP0939Lifter2.tyMotionStd.tyBtnJogDown.uiMaskRtStat));
	END_IF

	// Interlock Move Absolute
	IF p_bLifter2AxisErr = TRUE OR p_bLifter2PwrOn = FALSE OR p_bLifter2IsHomed = FALSE THEN

		fUIInRtStatOff(ADR(tyP0939Lifter2.tyMotionStd.tyBtnMovAbs.uiMaskRtStat));

		fUIInRtStatOff(ADR(tyP0939Lifter2.tyLifter.tyBtnGo.uiMaskRtStat));
		fUIInRtStatOff(ADR(tyP0939Lifter2.tyLifter.tyBtnNxtSlt.uiMaskRtStat));
		fUIInRtStatOff(ADR(tyP0939Lifter2.tyLifter.tyBtnPrevSlt.uiMaskRtStat));
		fUIInRtStatOff(ADR(tyP0939Lifter2.tyLifter.tyBtnGoLaneA.uiMaskRtStat));
		fUIInRtStatOff(ADR(tyP0939Lifter2.tyLifter.tyBtnGoLaneB.uiMaskRtStat));
		fUIInRtStatOff(ADR(tyP0939Lifter2.tyLifter.tyBtnGoLaneD_G.uiMaskRtStat));
		fUIInRtStatOff(ADR(tyP0939Lifter2.tyLifter.tyBtnGoLaneE_H.uiMaskRtStat));

	ELSE
		fUIInRtStatHide(ADR(tyP0939Lifter2.tyMotionStd.tyBtnMovAbs.uiMaskRtStat));

		fUIInRtStatHide(ADR(tyP0939Lifter2.tyLifter.tyBtnGo.uiMaskRtStat));
		fUIInRtStatHide(ADR(tyP0939Lifter2.tyLifter.tyBtnNxtSlt.uiMaskRtStat));
		fUIInRtStatHide(ADR(tyP0939Lifter2.tyLifter.tyBtnPrevSlt.uiMaskRtStat));
		fUIInRtStatHide(ADR(tyP0939Lifter2.tyLifter.tyBtnGoLaneA.uiMaskRtStat));
		fUIInRtStatHide(ADR(tyP0939Lifter2.tyLifter.tyBtnGoLaneB.uiMaskRtStat));
		fUIInRtStatHide(ADR(tyP0939Lifter2.tyLifter.tyBtnGoLaneD_G.uiMaskRtStat));
		fUIInRtStatHide(ADR(tyP0939Lifter2.tyLifter.tyBtnGoLaneE_H.uiMaskRtStat));

	END_IF

	//Interlock Limit Sensor
	IF tyP0939Lifter2.tyMotionStd.tyBtnDownLmtSen.bValue = TRUE THEN
		fUIInRtStatOff(ADR(tyP0939Lifter2.tyMotionStd.tyBtnJogDown.uiMaskRtStat));
	END_IF

	IF tyP0939Lifter2.tyMotionStd.tyBtnUpLmtSen.bValue = TRUE THEN
		fUIInRtStatOff(ADR(tyP0939Lifter2.tyMotionStd.tyBtnJogUp.uiMaskRtStat));
	END_IF

	// Interlock When Moving
	IF tyP0939Lifter2.tyMotionStd.tyBtnOrigin.bRtCompl = TRUE THEN

		fUIInRtStatOff(ADR(tyP0939Lifter2.tyMotionStd.tyBtnMovAbs.uiMaskRtStat));
		fUIInRtStatOff(ADR(tyP0939Lifter2.tyMotionStd.tyBtnMovRel.uiMaskRtStat));
		fUIInRtStatOff(ADR(tyP0939Lifter2.tyMotionStd.tyBtnJogUp.uiMaskRtStat));
		fUIInRtStatOff(ADR(tyP0939Lifter2.tyMotionStd.tyBtnJogDown.uiMaskRtStat));

		fUIInRtStatOff(ADR(tyP0939Lifter2.tyLifter.tyBtnGo.uiMaskRtStat));
		fUIInRtStatOff(ADR(tyP0939Lifter2.tyLifter.tyBtnPrevSlt.uiMaskRtStat));
		fUIInRtStatOff(ADR(tyP0939Lifter2.tyLifter.tyBtnNxtSlt.uiMaskRtStat));
		fUIInRtStatOff(ADR(tyP0939Lifter2.tyLifter.tyBtnGoLaneA.uiMaskRtStat));
		fUIInRtStatOff(ADR(tyP0939Lifter2.tyLifter.tyBtnGoLaneB.uiMaskRtStat));
		fUIInRtStatOff(ADR(tyP0939Lifter2.tyLifter.tyBtnGoLaneD_G.uiMaskRtStat));
		fUIInRtStatOff(ADR(tyP0939Lifter2.tyLifter.tyBtnGoLaneE_H.uiMaskRtStat));

	ELSIF tyP0939Lifter2.tyMotionStd.tyBtnMovAbs.bRtCompl = TRUE THEN

		fUIInRtStatOff(ADR(tyP0939Lifter2.tyMotionStd.tyBtnOrigin.uiMaskRtStat));
		fUIInRtStatOff(ADR(tyP0939Lifter2.tyMotionStd.tyBtnMovRel.uiMaskRtStat));
		fUIInRtStatOff(ADR(tyP0939Lifter2.tyMotionStd.tyBtnJogUp.uiMaskRtStat));
		fUIInRtStatOff(ADR(tyP0939Lifter2.tyMotionStd.tyBtnJogDown.uiMaskRtStat));

		fUIInRtStatOff(ADR(tyP0939Lifter2.tyLifter.tyBtnGo.uiMaskRtStat));
		fUIInRtStatOff(ADR(tyP0939Lifter2.tyLifter.tyBtnPrevSlt.uiMaskRtStat));
		fUIInRtStatOff(ADR(tyP0939Lifter2.tyLifter.tyBtnNxtSlt.uiMaskRtStat));
		fUIInRtStatOff(ADR(tyP0939Lifter2.tyLifter.tyBtnGoLaneA.uiMaskRtStat));
		fUIInRtStatOff(ADR(tyP0939Lifter2.tyLifter.tyBtnGoLaneB.uiMaskRtStat));
		fUIInRtStatOff(ADR(tyP0939Lifter2.tyLifter.tyBtnGoLaneD_G.uiMaskRtStat));
		fUIInRtStatOff(ADR(tyP0939Lifter2.tyLifter.tyBtnGoLaneE_H.uiMaskRtStat));

	ELSIF tyP0939Lifter2.tyMotionStd.tyBtnMovRel.bRtCompl = TRUE THEN

		fUIInRtStatOff(ADR(tyP0939Lifter2.tyMotionStd.tyBtnOrigin.uiMaskRtStat));
		fUIInRtStatOff(ADR(tyP0939Lifter2.tyMotionStd.tyBtnMovAbs.uiMaskRtStat));
		fUIInRtStatOff(ADR(tyP0939Lifter2.tyMotionStd.tyBtnJogUp.uiMaskRtStat));
		fUIInRtStatOff(ADR(tyP0939Lifter2.tyMotionStd.tyBtnJogDown.uiMaskRtStat));

		fUIInRtStatOff(ADR(tyP0939Lifter2.tyLifter.tyBtnGo.uiMaskRtStat));
		fUIInRtStatOff(ADR(tyP0939Lifter2.tyLifter.tyBtnNxtSlt.uiMaskRtStat));
		fUIInRtStatOff(ADR(tyP0939Lifter2.tyLifter.tyBtnPrevSlt.uiMaskRtStat));
		fUIInRtStatOff(ADR(tyP0939Lifter2.tyLifter.tyBtnGoLaneA.uiMaskRtStat));
		fUIInRtStatOff(ADR(tyP0939Lifter2.tyLifter.tyBtnGoLaneB.uiMaskRtStat));
		fUIInRtStatOff(ADR(tyP0939Lifter2.tyLifter.tyBtnGoLaneD_G.uiMaskRtStat));
		fUIInRtStatOff(ADR(tyP0939Lifter2.tyLifter.tyBtnGoLaneE_H.uiMaskRtStat));

	ELSIF tyP0939Lifter2.tyMotionStd.tyBtnJogDown.bRtCompl = TRUE OR tyP0939Lifter2.tyMotionStd.tyBtnJogDown.bValue = TRUE THEN
		fUIInRtStatOff(ADR(tyP0939Lifter2.tyMotionStd.tyBtnOrigin.uiMaskRtStat));
		fUIInRtStatOff(ADR(tyP0939Lifter2.tyMotionStd.tyBtnMovAbs.uiMaskRtStat));
		fUIInRtStatOff(ADR(tyP0939Lifter2.tyMotionStd.tyBtnMovRel.uiMaskRtStat));
		fUIInRtStatOff(ADR(tyP0939Lifter2.tyMotionStd.tyBtnJogUp.uiMaskRtStat));

		fUIInRtStatOff(ADR(tyP0939Lifter2.tyLifter.tyBtnGo.uiMaskRtStat));
		fUIInRtStatOff(ADR(tyP0939Lifter2.tyLifter.tyBtnNxtSlt.uiMaskRtStat));
		fUIInRtStatOff(ADR(tyP0939Lifter2.tyLifter.tyBtnPrevSlt.uiMaskRtStat));
		fUIInRtStatOff(ADR(tyP0939Lifter2.tyLifter.tyBtnGoLaneA.uiMaskRtStat));
		fUIInRtStatOff(ADR(tyP0939Lifter2.tyLifter.tyBtnGoLaneB.uiMaskRtStat));
		fUIInRtStatOff(ADR(tyP0939Lifter2.tyLifter.tyBtnGoLaneD_G.uiMaskRtStat));
		fUIInRtStatOff(ADR(tyP0939Lifter2.tyLifter.tyBtnGoLaneE_H.uiMaskRtStat));

	ELSIF tyP0939Lifter2.tyMotionStd.tyBtnJogUp.bRtCompl = TRUE OR tyP0939Lifter2.tyMotionStd.tyBtnJogUp.bValue = TRUE THEN
		fUIInRtStatOff(ADR(tyP0939Lifter2.tyMotionStd.tyBtnOrigin.uiMaskRtStat));
		fUIInRtStatOff(ADR(tyP0939Lifter2.tyMotionStd.tyBtnMovAbs.uiMaskRtStat));
		fUIInRtStatOff(ADR(tyP0939Lifter2.tyMotionStd.tyBtnMovRel.uiMaskRtStat));
		fUIInRtStatOff(ADR(tyP0939Lifter2.tyMotionStd.tyBtnJogDown.uiMaskRtStat));

		fUIInRtStatOff(ADR(tyP0939Lifter2.tyLifter.tyBtnGo.uiMaskRtStat));
		fUIInRtStatOff(ADR(tyP0939Lifter2.tyLifter.tyBtnNxtSlt.uiMaskRtStat));
		fUIInRtStatOff(ADR(tyP0939Lifter2.tyLifter.tyBtnPrevSlt.uiMaskRtStat));
		fUIInRtStatOff(ADR(tyP0939Lifter2.tyLifter.tyBtnGoLaneA.uiMaskRtStat));
		fUIInRtStatOff(ADR(tyP0939Lifter2.tyLifter.tyBtnGoLaneB.uiMaskRtStat));
		fUIInRtStatOff(ADR(tyP0939Lifter2.tyLifter.tyBtnGoLaneD_G.uiMaskRtStat));
		fUIInRtStatOff(ADR(tyP0939Lifter2.tyLifter.tyBtnGoLaneE_H.uiMaskRtStat));

	ELSIF tyP0939Lifter2.tyLifter.tyBtnGo.bRtCompl = TRUE THEN
		fUIInRtStatOff(ADR(tyP0939Lifter2.tyMotionStd.tyBtnOrigin.uiMaskRtStat));
		fUIInRtStatOff(ADR(tyP0939Lifter2.tyMotionStd.tyBtnMovAbs.uiMaskRtStat));
		fUIInRtStatOff(ADR(tyP0939Lifter2.tyMotionStd.tyBtnMovRel.uiMaskRtStat));
		fUIInRtStatOff(ADR(tyP0939Lifter2.tyMotionStd.tyBtnJogUp.uiMaskRtStat));
		fUIInRtStatOff(ADR(tyP0939Lifter2.tyMotionStd.tyBtnJogDown.uiMaskRtStat));

		fUIInRtStatOff(ADR(tyP0939Lifter2.tyLifter.tyBtnNxtSlt.uiMaskRtStat));
		fUIInRtStatOff(ADR(tyP0939Lifter2.tyLifter.tyBtnPrevSlt.uiMaskRtStat));
		fUIInRtStatOff(ADR(tyP0939Lifter2.tyLifter.tyBtnGoLaneA.uiMaskRtStat));
		fUIInRtStatOff(ADR(tyP0939Lifter2.tyLifter.tyBtnGoLaneB.uiMaskRtStat));
		fUIInRtStatOff(ADR(tyP0939Lifter2.tyLifter.tyBtnGoLaneD_G.uiMaskRtStat));
		fUIInRtStatOff(ADR(tyP0939Lifter2.tyLifter.tyBtnGoLaneE_H.uiMaskRtStat));

	ELSIF tyP0939Lifter2.tyLifter.tyBtnNxtSlt.bRtCompl = TRUE THEN
		fUIInRtStatOff(ADR(tyP0939Lifter2.tyMotionStd.tyBtnOrigin.uiMaskRtStat));
		fUIInRtStatOff(ADR(tyP0939Lifter2.tyMotionStd.tyBtnMovAbs.uiMaskRtStat));
		fUIInRtStatOff(ADR(tyP0939Lifter2.tyMotionStd.tyBtnMovRel.uiMaskRtStat));
		fUIInRtStatOff(ADR(tyP0939Lifter2.tyMotionStd.tyBtnJogUp.uiMaskRtStat));
		fUIInRtStatOff(ADR(tyP0939Lifter2.tyMotionStd.tyBtnJogDown.uiMaskRtStat));

		fUIInRtStatOff(ADR(tyP0939Lifter2.tyLifter.tyBtnGo.uiMaskRtStat));
		fUIInRtStatOff(ADR(tyP0939Lifter2.tyLifter.tyBtnPrevSlt.uiMaskRtStat));
		fUIInRtStatOff(ADR(tyP0939Lifter2.tyLifter.tyBtnGoLaneA.uiMaskRtStat));
		fUIInRtStatOff(ADR(tyP0939Lifter2.tyLifter.tyBtnGoLaneB.uiMaskRtStat));
		fUIInRtStatOff(ADR(tyP0939Lifter2.tyLifter.tyBtnGoLaneD_G.uiMaskRtStat));
		fUIInRtStatOff(ADR(tyP0939Lifter2.tyLifter.tyBtnGoLaneE_H.uiMaskRtStat));

	ELSIF tyP0939Lifter2.tyLifter.tyBtnPrevSlt.bRtCompl = TRUE THEN
		fUIInRtStatOff(ADR(tyP0939Lifter2.tyMotionStd.tyBtnOrigin.uiMaskRtStat));
		fUIInRtStatOff(ADR(tyP0939Lifter2.tyMotionStd.tyBtnMovAbs.uiMaskRtStat));
		fUIInRtStatOff(ADR(tyP0939Lifter2.tyMotionStd.tyBtnMovRel.uiMaskRtStat));
		fUIInRtStatOff(ADR(tyP0939Lifter2.tyMotionStd.tyBtnJogUp.uiMaskRtStat));
		fUIInRtStatOff(ADR(tyP0939Lifter2.tyMotionStd.tyBtnJogDown.uiMaskRtStat));

		fUIInRtStatOff(ADR(tyP0939Lifter2.tyLifter.tyBtnGo.uiMaskRtStat));
		fUIInRtStatOff(ADR(tyP0939Lifter2.tyLifter.tyBtnNxtSlt.uiMaskRtStat));
		fUIInRtStatOff(ADR(tyP0939Lifter2.tyLifter.tyBtnGoLaneA.uiMaskRtStat));
		fUIInRtStatOff(ADR(tyP0939Lifter2.tyLifter.tyBtnGoLaneB.uiMaskRtStat));
		fUIInRtStatOff(ADR(tyP0939Lifter2.tyLifter.tyBtnGoLaneD_G.uiMaskRtStat));
		fUIInRtStatOff(ADR(tyP0939Lifter2.tyLifter.tyBtnGoLaneE_H.uiMaskRtStat));

	ELSIF tyP0939Lifter2.tyLifter.tyBtnGoLaneA.bRtCompl = TRUE THEN
		fUIInRtStatOff(ADR(tyP0939Lifter2.tyMotionStd.tyBtnOrigin.uiMaskRtStat));
		fUIInRtStatOff(ADR(tyP0939Lifter2.tyMotionStd.tyBtnMovAbs.uiMaskRtStat));
		fUIInRtStatOff(ADR(tyP0939Lifter2.tyMotionStd.tyBtnMovRel.uiMaskRtStat));
		fUIInRtStatOff(ADR(tyP0939Lifter2.tyMotionStd.tyBtnJogUp.uiMaskRtStat));
		fUIInRtStatOff(ADR(tyP0939Lifter2.tyMotionStd.tyBtnJogDown.uiMaskRtStat));

		fUIInRtStatOff(ADR(tyP0939Lifter2.tyLifter.tyBtnGo.uiMaskRtStat));
		fUIInRtStatOff(ADR(tyP0939Lifter2.tyLifter.tyBtnNxtSlt.uiMaskRtStat));
		fUIInRtStatOff(ADR(tyP0939Lifter2.tyLifter.tyBtnPrevSlt.uiMaskRtStat));
		fUIInRtStatOff(ADR(tyP0939Lifter2.tyLifter.tyBtnGoLaneB.uiMaskRtStat));
		fUIInRtStatOff(ADR(tyP0939Lifter2.tyLifter.tyBtnGoLaneE_H.uiMaskRtStat));

	ELSIF tyP0939Lifter2.tyLifter.tyBtnGoLaneB.bRtCompl = TRUE THEN
		fUIInRtStatOff(ADR(tyP0939Lifter2.tyMotionStd.tyBtnOrigin.uiMaskRtStat));
		fUIInRtStatOff(ADR(tyP0939Lifter2.tyMotionStd.tyBtnMovAbs.uiMaskRtStat));
		fUIInRtStatOff(ADR(tyP0939Lifter2.tyMotionStd.tyBtnMovRel.uiMaskRtStat));
		fUIInRtStatOff(ADR(tyP0939Lifter2.tyMotionStd.tyBtnJogUp.uiMaskRtStat));
		fUIInRtStatOff(ADR(tyP0939Lifter2.tyMotionStd.tyBtnJogDown.uiMaskRtStat));

		fUIInRtStatOff(ADR(tyP0939Lifter2.tyLifter.tyBtnGo.uiMaskRtStat));
		fUIInRtStatOff(ADR(tyP0939Lifter2.tyLifter.tyBtnNxtSlt.uiMaskRtStat));
		fUIInRtStatOff(ADR(tyP0939Lifter2.tyLifter.tyBtnPrevSlt.uiMaskRtStat));
		fUIInRtStatOff(ADR(tyP0939Lifter2.tyLifter.tyBtnGoLaneA.uiMaskRtStat));
		fUIInRtStatOff(ADR(tyP0939Lifter2.tyLifter.tyBtnGoLaneD_G.uiMaskRtStat));

	END_IF

	//Axis Error
	IF tyP0939Lifter2.tyMotionStd.tyBtnPwr.bRtCompl = TRUE THEN
		fUIInRtStatOff(ADR(tyP0939Lifter2.tyMotionStd.tyBtnRst.uiMaskRtStat));
	ELSE
		fUIInRtStatHide(ADR(tyP0939Lifter2.tyMotionStd.tyBtnRst.uiMaskRtStat));
	END_IF

	//Next Slot
	IF p_diLifter2CurrSltA >= p_tyProdRcpCurrRcp0.diMaxSltValue THEN
		fUIInRtStatOff(ADR(tyP0939Lifter2.tyLifter.tyBtnNxtSlt.uiMaskRtStat));
	END_IF

	//Previous Slot
	IF p_diLifter2CurrSltA <= p_tyProdRcpCurrRcp0.diMinSltValue THEN
		fUIInRtStatOff(ADR(tyP0939Lifter2.tyLifter.tyBtnPrevSlt.uiMaskRtStat));
	END_IF

END_ACTION
```

#### Act_OptP0939UpdtDat.st
```iecst
ACTION Act_OptP0939UpdtDat:

	tyP0939Lifter2.tyMotionStd.tyNumCurrPos.diValue			:= p_diLifter2ActualPos;
	tyP0939Lifter2.tyMotionStd.tyNumErrCode.diValue			:= UDINT_TO_DINT(p_udiLifter2AxisErrID);
	tyP0939Lifter2.tyMotionStd.tyBitmapPwr.usiValueIdx		:= BOOL_TO_USINT(p_bLifter2PwrOn);
	tyP0939Lifter2.tyMotionStd.tyBitmapRst.usiValueIdx		:= BOOL_TO_USINT(NOT p_bLifter2AxisErr);
	tyP0939Lifter2.tyMotionStd.tyBitmapOrigin.usiValueIdx	:= BOOL_TO_USINT(p_bLifter2IsHomed);
	tyP0939Lifter2.tyMotionStd.tyBtnUpLmtSen.bValue			:= p_bLifter2UpSen;
	tyP0939Lifter2.tyMotionStd.tyBtnDownLmtSen.bValue		:= p_bLifter2DownSen;

	//Machine Bitmap
	IF p_bLifter2IsHomed = TRUE THEN
		IF p_diLifter2ActualPos <= (p_tyNtParamCurr.tyUILifterTargetPos.diMax / 3) THEN
			tyP0939Lifter2.tyMotionStd.tyBitmapMc.uiValueIdx 	:= 2;
		ELSIF p_diLifter2ActualPos <= (p_tyNtParamCurr.tyUILifterTargetPos.diMax / 3 * 2) THEN
			tyP0939Lifter2.tyMotionStd.tyBitmapMc.uiValueIdx 	:= 3;
		ELSE
			tyP0939Lifter2.tyMotionStd.tyBitmapMc.uiValueIdx 	:= 4;
		END_IF
	ELSE
		tyP0939Lifter2.tyMotionStd.tyBitmapMc.uiValueIdx	:= 2;
	END_IF

//	IF p_tyNtParamCurr.eProjMag = ULMagTriple THEN
//		tyP0939Lifter2.tyMotionStd.tyBitmapMc.uiValueIdx	:= tyP0939Lifter2.tyMotionStd.tyBitmapMc.uiValueIdx + 100;
//	END_IF

	IF p_tyNtParamCurr.eProjMag = ULMagDual THEN
		IF p_tyNtParamCurr.bProjLifterMagPlatform AND p_tyNtParamCurr.bUIConvDirRL THEN
			IF 	tyP0939Lifter2.tyMotionStd.tyBitmapMc.uiValueIdx < 700 THEN
				tyP0939Lifter2.tyMotionStd.tyBitmapMc.uiValueIdx	:= tyP0939Lifter2.tyMotionStd.tyBitmapMc.uiValueIdx + 700;
			END_IF
		ELSIF p_tyNtParamCurr.bProjLifterMagPlatform THEN
			IF p_tyNtParamCurr.bProjMagConvLane2Prep = FALSE THEN
				IF 	tyP0939Lifter2.tyMotionStd.tyBitmapMc.uiValueIdx < 600 THEN
					tyP0939Lifter2.tyMotionStd.tyBitmapMc.uiValueIdx	:= tyP0939Lifter2.tyMotionStd.tyBitmapMc.uiValueIdx + 600;
				END_IF
			ELSE
				IF 	tyP0939Lifter2.tyMotionStd.tyBitmapMc.uiValueIdx < 903 THEN //Lifter 2 - 905,906,907
					tyP0939Lifter2.tyMotionStd.tyBitmapMc.uiValueIdx	:= tyP0939Lifter2.tyMotionStd.tyBitmapMc.uiValueIdx + 903;
				END_IF
			END_IF
		ELSIF p_tyNtParamCurr.bMagAutoVerifyPrep = FALSE THEN
			IF 	tyP0939Lifter2.tyMotionStd.tyBitmapMc.uiValueIdx < 100 THEN
				tyP0939Lifter2.tyMotionStd.tyBitmapMc.uiValueIdx	:= tyP0939Lifter2.tyMotionStd.tyBitmapMc.uiValueIdx + 300;
			END_IF
		ELSE
			IF 	tyP0939Lifter2.tyMotionStd.tyBitmapMc.uiValueIdx < 300 THEN
				tyP0939Lifter2.tyMotionStd.tyBitmapMc.uiValueIdx	:= tyP0939Lifter2.tyMotionStd.tyBitmapMc.uiValueIdx + 300;
			END_IF
		END_IF
	ELSIF p_tyNtParamCurr.eProjMag = ULMagTriple THEN
		IF p_tyNtParamCurr.bProjLifterMagPlatform AND p_tyNtParamCurr.bUIConvDirRL THEN
			IF 	tyP0939Lifter2.tyMotionStd.tyBitmapMc.uiValueIdx < 800 THEN
				tyP0939Lifter2.tyMotionStd.tyBitmapMc.uiValueIdx	:= tyP0939Lifter2.tyMotionStd.tyBitmapMc.uiValueIdx + 800;
			END_IF
		ELSIF p_tyNtParamCurr.bProjLifterMagPlatform THEN
			IF tyP0939Lifter2.tyMotionStd.tyBitmapMc.uiValueIdx < 500 THEN
				tyP0939Lifter2.tyMotionStd.tyBitmapMc.uiValueIdx	:= tyP0939Lifter2.tyMotionStd.tyBitmapMc.uiValueIdx + 500;
			END_IF
		ELSIF p_tyNtParamCurr.bMagAutoVerifyPrep = TRUE AND p_tyNtParamCurr.bProjMotorizedPusherPrep = FALSE THEN
			IF 	tyP0939Lifter2.tyMotionStd.tyBitmapMc.uiValueIdx < 200 THEN
				tyP0939Lifter2.tyMotionStd.tyBitmapMc.uiValueIdx	:= tyP0939Lifter2.tyMotionStd.tyBitmapMc.uiValueIdx + 200;
			END_IF
		ELSIF  p_tyNtParamCurr.bMagAutoVerifyPrep = FALSE AND p_tyNtParamCurr.bProjMotorizedPusherPrep = TRUE THEN
			IF 	tyP0939Lifter2.tyMotionStd.tyBitmapMc.uiValueIdx < 400 THEN
				tyP0939Lifter2.tyMotionStd.tyBitmapMc.uiValueIdx	:= tyP0939Lifter2.tyMotionStd.tyBitmapMc.uiValueIdx + 400;
			END_IF
		END_IF
	END_IF

END_ACTION
```

#### Act_OptP0939Keypad.st
```iecst
ACTION Act_OptP0939Keypad:

	IF fUIOutRtStatTPIsOpen(ADR(tyP0939Lifter2.tyMotionStd.tyNumTargetPos.uiRtStat)) = TRUE THEN
		tyProperty.tyKeypad.tyStringTitle.sKeypadTitle	:= tyP0939Lifter2.tyMotionStd.tyNumTargetPos.sKeypadTitle;

	ELSIF fUIOutRtStatTPIsOpen(ADR(tyP0939Lifter2.tyMotionStd.tyNumStepSize.uiRtStat)) = TRUE THEN
		tyProperty.tyKeypad.tyStringTitle.sKeypadTitle	:= tyP0939Lifter2.tyMotionStd.tyNumStepSize.sKeypadTitle;

	ELSIF fUIOutRtStatTPIsOpen(ADR(tyP0939Lifter2.tyMotionStd.tyNumNomSpd.uiRtStat)) = TRUE THEN
		tyProperty.tyKeypad.tyStringTitle.sKeypadTitle	:= tyP0939Lifter2.tyMotionStd.tyNumNomSpd.sKeypadTitle;

	ELSIF fUIOutRtStatTPIsOpen(ADR(tyP0939Lifter2.tyMotionStd.tyNumSlwSpd.uiRtStat)) = TRUE THEN
		tyProperty.tyKeypad.tyStringTitle.sKeypadTitle	:= tyP0939Lifter2.tyMotionStd.tyNumSlwSpd.sKeypadTitle;

	ELSIF fUIOutRtStatTPIsOpen(ADR(tyP0939Lifter2.tyLifter.tyNumNewSlt.uiRtStat)) = TRUE THEN
		tyProperty.tyKeypad.tyStringTitle.sKeypadTitle	:= tyP0939Lifter2.tyLifter.tyNumNewSlt.sKeypadTitle;

	ELSIF fUIOutRtStatTPIsOpen(ADR(tyP0939Lifter2.tyLifter.tyNumMagPos.uiRtStat)) = TRUE THEN
		tyProperty.tyKeypad.tyStringTitle.sKeypadTitle	:= tyP0939Lifter2.tyLifter.tyNumMagPos.sKeypadTitle;

	END_IF

END_ACTION
```

#### Act_OptP0939RstMnl.st
```iecst
ACTION Act_OptP0939RstMnl:

	IF EDGEPOS((bManualMod = FALSE) OR (p_eLifter2Status = Error)) THEN

		eLifter2Act	:= LifterActIdle;

		bJogSlow				:= FALSE;
		bJogFast				:= FALSE;
		fbJogSlowToFastDlyTm.IN	:= FALSE;

		tyP0939Lifter2.tyLifter.tyBtnGo.bRtCompl					:= FALSE;
		tyP0939Lifter2.tyLifter.tyBtnNxtSlt.bRtCompl				:= FALSE;
		tyP0939Lifter2.tyLifter.tyBtnPrevSlt.bRtCompl			:= FALSE;
		tyP0939Lifter2.tyLifter.tyBtnGoLaneA.bRtCompl			:= FALSE;
		tyP0939Lifter2.tyLifter.tyBtnGoLaneB.bRtCompl			:= FALSE;
		tyP0939Lifter2.tyLifter.tyBtnGoLaneD_G.bRtCompl			:= FALSE;
		tyP0939Lifter2.tyLifter.tyBtnGoLaneE_H.bRtCompl			:= FALSE;

		tyP0939Lifter2.tyLifter.tyBtnGo.bValue					:= FALSE;
		tyP0939Lifter2.tyLifter.tyBtnNxtSlt.bValue				:= FALSE;
		tyP0939Lifter2.tyLifter.tyBtnPrevSlt.bValue				:= FALSE;
		tyP0939Lifter2.tyLifter.tyBtnGoLaneA.bValue				:= FALSE;
		tyP0939Lifter2.tyLifter.tyBtnGoLaneB.bValue				:= FALSE;
		tyP0939Lifter2.tyLifter.tyBtnGoLaneD_G.bValue				:= FALSE;
		tyP0939Lifter2.tyLifter.tyBtnGoLaneE_H.bValue				:= FALSE;

		tyP0939Lifter2.tyLifter.tyBtnGo.bRtLk					:= FALSE;
		tyP0939Lifter2.tyLifter.tyBtnNxtSlt.bRtLk				:= FALSE;
		tyP0939Lifter2.tyLifter.tyBtnPrevSlt.bRtLk				:= FALSE;
		tyP0939Lifter2.tyLifter.tyBtnGoLaneA.bRtLk				:= FALSE;
		tyP0939Lifter2.tyLifter.tyBtnGoLaneB.bRtLk				:= FALSE;
		tyP0939Lifter2.tyLifter.tyBtnGoLaneD_G.bRtLk				:= FALSE;
		tyP0939Lifter2.tyLifter.tyBtnGoLaneE_H.bRtLk				:= FALSE;

		tyP0939Lifter2.tyLifter.tyBtnGo.uiMaskRtStat.0			:= FALSE;
		tyP0939Lifter2.tyLifter.tyBtnNxtSlt.uiMaskRtStat.0		:= FALSE;
		tyP0939Lifter2.tyLifter.tyBtnPrevSlt.uiMaskRtStat.0		:= FALSE;
		tyP0939Lifter2.tyLifter.tyBtnGoLaneA.uiMaskRtStat.0		:= FALSE;
		tyP0939Lifter2.tyLifter.tyBtnGoLaneB.uiMaskRtStat.0		:= FALSE;
		tyP0939Lifter2.tyLifter.tyBtnGoLaneD_G.uiMaskRtStat.0		:= FALSE;
		tyP0939Lifter2.tyLifter.tyBtnGoLaneE_H.uiMaskRtStat.0		:= FALSE;

		tyP0939Lifter2.tyMotionStd.tyBtnPwr.bRtCompl				:= FALSE;
		tyP0939Lifter2.tyMotionStd.tyBtnStop.bRtCompl			:= FALSE;
		tyP0939Lifter2.tyMotionStd.tyBtnOrigin.bRtCompl			:= FALSE;
		tyP0939Lifter2.tyMotionStd.tyBtnRst.bRtCompl				:= FALSE;
		tyP0939Lifter2.tyMotionStd.tyBtnMovAbs.bRtCompl			:= FALSE;
		tyP0939Lifter2.tyMotionStd.tyBtnMovRel.bRtCompl			:= FALSE;
		tyP0939Lifter2.tyMotionStd.tyBtnJogUp.bRtCompl			:= FALSE;
		tyP0939Lifter2.tyMotionStd.tyBtnJogDown.bRtCompl			:= FALSE;

		tyP0939Lifter2.tyMotionStd.tyBtnPwr.bValue				:= FALSE;
		tyP0939Lifter2.tyMotionStd.tyBtnStop.bValue				:= TRUE;
		tyP0939Lifter2.tyMotionStd.tyBtnOrigin.bValue			:= FALSE;
		tyP0939Lifter2.tyMotionStd.tyBtnRst.bValue				:= FALSE;
		tyP0939Lifter2.tyMotionStd.tyBtnMovAbs.bValue			:= FALSE;
		tyP0939Lifter2.tyMotionStd.tyBtnMovRel.bValue			:= FALSE;
		tyP0939Lifter2.tyMotionStd.tyBtnJogUp.bValue				:= FALSE;
		tyP0939Lifter2.tyMotionStd.tyBtnJogDown.bValue			:= FALSE;

		tyP0939Lifter2.tyMotionStd.tyBtnPwr.bRtLk				:= FALSE;
		tyP0939Lifter2.tyMotionStd.tyBtnStop.bRtLk				:= TRUE;
		tyP0939Lifter2.tyMotionStd.tyBtnOrigin.bRtLk				:= FALSE;
		tyP0939Lifter2.tyMotionStd.tyBtnRst.bRtLk				:= FALSE;
		tyP0939Lifter2.tyMotionStd.tyBtnMovAbs.bRtLk				:= FALSE;
		tyP0939Lifter2.tyMotionStd.tyBtnMovRel.bRtLk				:= FALSE;
		tyP0939Lifter2.tyMotionStd.tyBtnJogUp.bRtLk				:= FALSE;
		tyP0939Lifter2.tyMotionStd.tyBtnJogDown.bRtLk			:= FALSE;

		tyP0939Lifter2.tyMotionStd.tyBtnPwr.uiMaskRtStat			:= TRUE;
		tyP0939Lifter2.tyMotionStd.tyBtnOrigin.uiMaskRtStat		:= FALSE;
		tyP0939Lifter2.tyMotionStd.tyBtnRst.uiMaskRtStat			:= TRUE;
		tyP0939Lifter2.tyMotionStd.tyBtnMovAbs.uiMaskRtStat		:= FALSE;
		tyP0939Lifter2.tyMotionStd.tyBtnMovRel.uiMaskRtStat		:= FALSE;
		tyP0939Lifter2.tyMotionStd.tyBtnJogUp.uiMaskRtStat		:= FALSE;
		tyP0939Lifter2.tyMotionStd.tyBtnJogDown.uiMaskRtStat		:= FALSE;

	END_IF

	eInShutterAct	:= PneuActIdle;
	eOutShutterAct	:= PneuActIdle;

	tyP0939Lifter2.tyInOutletShutterFB.tyBtnClose.bRtCompl	:= FALSE;
	tyP0939Lifter2.tyInOutletShutterFB.tyBtnClose.bValue	:= FALSE;
	tyP0939Lifter2.tyInOutletShutterFB.tyBtnOpen.bRtCompl	:= FALSE;
	tyP0939Lifter2.tyInOutletShutterFB.tyBtnOpen.bValue	:= FALSE;

END_ACTION
```

#### Act_EntP0940Disp.st
```iecst
ACTION Act_EntP0940Disp:

	//Access Address
	p_tyC0005Main ACCESS ADR(tyCommon.tyMain);

	p_tyC0007Notif ACCESS ADR(tyCommon.tyNotif);

	p_tyC0008MsgBox ACCESS ADR(tyP0940CommCtrl.tyMsgBoxHide);

	p_tyC0009Info ACCESS ADR(tyCommon.tyInfo);

	p_tyP0940CommCtrlUSSMEMAA ACCESS ADR(tyP0940CommCtrl.tyUSSMEMAA);
	p_tyP0940CommCtrlUSSMEMAB ACCESS ADR(tyP0940CommCtrl.tyUSSMEMAB);
	p_tyP0940CommCtrlSOT ACCESS ADR(tyP0940CommCtrl.tySOT);
	p_tyP0940CommDMCRFID ACCESS ADR(tyP0940CommCtrl.tyDMCRFID);
	//Upstream Line A
	IF p_tyMcParamCurr.tyUSCommASMEMA.bStatSigSetGd = TRUE THEN
		tyP0940CommCtrl.tyUSSMEMAA.tyBtnUBAStat.usiTxtIdx	:= 0;
	ELSE
		tyP0940CommCtrl.tyUSSMEMAA.tyBtnUBAStat.usiTxtIdx	:= 1;
	END_IF

	tyP0940CommCtrl.tyUSSMEMAA.tyBtnUBAStat.uiRtStat.0	:= NOT(p_tyMcParamCurr.tyUSCommASMEMA.eSelection = SMEMASelIPC9851Ext);

	//Upstream Line B
	IF p_tyMcParamCurr.tyUSCommBSMEMA.bStatSigSetGd = TRUE THEN
		tyP0940CommCtrl.tyUSSMEMAB.tyBtnUBAStat.usiTxtIdx	:= 0;
	ELSE
		tyP0940CommCtrl.tyUSSMEMAB.tyBtnUBAStat.usiTxtIdx	:= 1;
	END_IF

	tyP0940CommCtrl.tyUSSMEMAB.tyBtnUBAStat.uiRtStat.0	:= NOT(p_tyMcParamCurr.tyUSCommBSMEMA.eSelection = SMEMASelIPC9851Ext);

	CASE p_tyMcParamCurr.eAGVComProtocol OF
		McSetAGVCommOPCUA:
			tyP0940CommCtrl.tySOT.tyTxtAIVCommProtocol.usiValueIdx := 0;

		McSetAGVCommHardIO:
			tyP0940CommCtrl.tySOT.tyTxtAIVCommProtocol.usiValueIdx := 1;

		McSetAGVCommDisabled:
			tyP0940CommCtrl.tySOT.tyTxtAIVCommProtocol.usiValueIdx := 2;

	END_CASE

END_ACTION
```

#### Act_OptP0940FullMask.st
```iecst
ACTION Act_OptP0940FullMask:

	IF eCurrPage = UIP0940CommCtrl THEN

		IF p_tyDI.bEStopSig = FALSE THEN
			p_tyC0002FullMask ACCESS ADR(tyP0940CommCtrl.tyFullMaskEStop);

		ELSIF p_tyDI.bCoverSWSig = FALSE THEN
			p_tyC0002FullMask ACCESS ADR(tyP0940CommCtrl.tyFullMaskCWSig);

		ELSIF p_tyDI.bSafetyRlySig = FALSE THEN
			p_tyC0002FullMask ACCESS ADR(tyP0940CommCtrl.tyFullMaskSafetyRly);

		ELSE
			p_tyC0002FullMask ACCESS ADR(tyP0940CommCtrl.tyFullMaskHide);

		END_IF

	END_IF

END_ACTION
```

#### Act_OptP0940ReadDI.st
```iecst
ACTION Act_OptP0940ReadDI:

		tyP0940CommCtrl.tyUSSMEMAA.tyBtnUBA.bValue		:= p_tyDI.bUBAA;
		tyP0940CommCtrl.tyUSSMEMAA.tyBtnUBAStat.bValue	:= p_tyDI.bUBAAStat;
		tyP0940CommCtrl.tyUSSMEMAB.tyBtnUBA.bValue		:= p_tyDI.bUBAB;
		tyP0940CommCtrl.tyUSSMEMAB.tyBtnUBAStat.bValue	:= p_tyDI.bUBABStat;

	IF p_tyNtParamCurr.bProjSOTSensorPrep THEN
//		CASE p_tyMcParamCurr.eAGVComProtocol OF
//			McSetAGVCommHardIO, :
				tyP0940CommCtrl.tySOT.tyBtnAIVRcv1.bValue		:= p_tyDI.bSOT1Receive;
				tyP0940CommCtrl.tySOT.tyBtnAIVErr1.bValue		:= p_tyDI.bSOT1AIVError;
				tyP0940CommCtrl.tySOT.tyBtnAIVRdy1.bValue		:= p_tyDI.bSOT1AIVReady;
				tyP0940CommCtrl.tySOT.tyBtnAIVAvail1.bValue		:= p_tyDI.bSOT1AIVAvailable;
				tyP0940CommCtrl.tySOT.tyBtnAIVSLarge1.bValue	:= p_tyDI.bSOT1AIVSizeLarge;

				tyP0940CommCtrl.tySOT.tyBtnAIVRcv2.bValue		:= p_tyDI.bSOT2Receive;
				tyP0940CommCtrl.tySOT.tyBtnAIVErr2.bValue		:= p_tyDI.bSOT2AIVError;
				tyP0940CommCtrl.tySOT.tyBtnAIVRdy2.bValue		:= p_tyDI.bSOT2AIVReady;
				tyP0940CommCtrl.tySOT.tyBtnAIVAvail2.bValue		:= p_tyDI.bSOT2AIVAvailable;
				tyP0940CommCtrl.tySOT.tyBtnAIVSLarge2.bValue	:= p_tyDI.bSOT2AIVSizeLarge;

				tyP0940CommCtrl.tySOT.tyBtnAIVRcv3.bValue		:= p_tyDI.bSOT3Receive;
				tyP0940CommCtrl.tySOT.tyBtnAIVErr3.bValue		:= p_tyDI.bSOT3AIVError;
				tyP0940CommCtrl.tySOT.tyBtnAIVRdy3.bValue		:= p_tyDI.bSOT3AIVReady;
				tyP0940CommCtrl.tySOT.tyBtnAIVAvail3.bValue		:= p_tyDI.bSOT3AIVAvailable;
				tyP0940CommCtrl.tySOT.tyBtnAIVSLarge3.bValue	:= p_tyDI.bSOT3AIVSizeLarge;

				tyP0940CommCtrl.tySOT.tyBtnAIVRcv4.bValue		:= p_tyDI.bSOT4Receive;
				tyP0940CommCtrl.tySOT.tyBtnAIVErr4.bValue		:= p_tyDI.bSOT4AIVError;
				tyP0940CommCtrl.tySOT.tyBtnAIVRdy4.bValue		:= p_tyDI.bSOT4AIVReady;
				tyP0940CommCtrl.tySOT.tyBtnAIVAvail4.bValue		:= p_tyDI.bSOT4AIVAvailable;
				tyP0940CommCtrl.tySOT.tyBtnAIVSLarge4.bValue	:= p_tyDI.bSOT4AIVSizeLarge;

				tyP0940CommCtrl.tySOT.tyBtnFleetMgrActive.bValue := p_tyDI.bFleetManagerReady OR p_tyTagFromMes.bActive;

//			McSetAGVCommOPCUA:
//
//				tyP0940CommCtrl.tySOT.tyBtnAIVErr1.bValue		:= p_tyTagFromMes.tyTagStatOfPlatforms[1].bError;
//				tyP0940CommCtrl.tySOT.tyBtnAIVRdy1.bValue		:= p_tyTagFromMes.tyTagStatOfPlatforms[1].bReady;
//				tyP0940CommCtrl.tySOT.tyBtnAIVAvail1.bValue		:= p_tyTagFromMes.tyTagStatOfPlatforms[1].bAvailable;
//				tyP0940CommCtrl.tySOT.tyBtnAIVSLarge1.bValue	:= p_tyTagFromMes.tyTagStatOfPlatforms[1].bSizeLarge;
//
//				tyP0940CommCtrl.tySOT.tyBtnAIVErr2.bValue		:= p_tyTagFromMes.tyTagStatOfPlatforms[2].bError;
//				tyP0940CommCtrl.tySOT.tyBtnAIVRdy2.bValue		:= p_tyTagFromMes.tyTagStatOfPlatforms[2].bReady;
//				tyP0940CommCtrl.tySOT.tyBtnAIVAvail2.bValue		:= p_tyTagFromMes.tyTagStatOfPlatforms[2].bAvailable;
//				tyP0940CommCtrl.tySOT.tyBtnAIVSLarge2.bValue	:= p_tyTagFromMes.tyTagStatOfPlatforms[2].bSizeLarge;
//
//				tyP0940CommCtrl.tySOT.tyBtnAIVErr3.bValue		:= p_tyTagFromMes.tyTagStatOfPlatforms[3].bError;
//				tyP0940CommCtrl.tySOT.tyBtnAIVRdy3.bValue		:= p_tyTagFromMes.tyTagStatOfPlatforms[3].bReady;
//				tyP0940CommCtrl.tySOT.tyBtnAIVAvail3.bValue		:= p_tyTagFromMes.tyTagStatOfPlatforms[3].bAvailable;
//				tyP0940CommCtrl.tySOT.tyBtnAIVSLarge3.bValue	:= p_tyTagFromMes.tyTagStatOfPlatforms[3].bSizeLarge;
//
//				tyP0940CommCtrl.tySOT.tyBtnAIVErr4.bValue		:= p_tyTagFromMes.tyTagStatOfPlatforms[4].bError;
//				tyP0940CommCtrl.tySOT.tyBtnAIVRdy4.bValue		:= p_tyTagFromMes.tyTagStatOfPlatforms[4].bReady;
//				tyP0940CommCtrl.tySOT.tyBtnAIVAvail4.bValue		:= p_tyTagFromMes.tyTagStatOfPlatforms[4].bAvailable;
//				tyP0940CommCtrl.tySOT.tyBtnAIVSLarge4.bValue	:= p_tyTagFromMes.tyTagStatOfPlatforms[4].bSizeLarge;
//
//				tyP0940CommCtrl.tySOT.tyBtnFleetMgrActive.bValue := p_tyTagFromMes.bActive;

//		END_CASE
	ELSIF p_tyMcParamCurr.eAGVComProtocol = McSetAGVCommHardIO AND p_tyNtParamCurr.bProjSOTSensorPrep = FALSE THEN
		tyP0940CommCtrl.tySOT.tyBtnAIVRcv1.bValue		:= p_tyDI.bSOT1Receive;
		tyP0940CommCtrl.tySOT.tyBtnAIVErr1.bValue		:= p_tyDI.bSOT1AIVError;
		tyP0940CommCtrl.tySOT.tyBtnAIVRdy1.bValue		:= p_tyDI.bSOT1AIVReady;
		tyP0940CommCtrl.tySOT.tyBtnAIVAvail1.bValue		:= p_tyDI.bSOT1AIVAvailable;
		tyP0940CommCtrl.tySOT.tyBtnAIVSLarge1.bValue	:= p_tyDI.bSOT1AIVSizeLarge;

		tyP0940CommCtrl.tySOT.tyBtnAIVRcv2.bValue		:= p_tyDI.bSOT2Receive;
		tyP0940CommCtrl.tySOT.tyBtnAIVErr2.bValue		:= p_tyDI.bSOT2AIVError;
		tyP0940CommCtrl.tySOT.tyBtnAIVRdy2.bValue		:= p_tyDI.bSOT2AIVReady;
		tyP0940CommCtrl.tySOT.tyBtnAIVAvail2.bValue		:= p_tyDI.bSOT2AIVAvailable;
		tyP0940CommCtrl.tySOT.tyBtnAIVSLarge2.bValue	:= p_tyDI.bSOT2AIVSizeLarge;

		tyP0940CommCtrl.tySOT.tyBtnAIVRcv3.bValue		:= p_tyDI.bSOT3Receive;
		tyP0940CommCtrl.tySOT.tyBtnAIVErr3.bValue		:= p_tyDI.bSOT3AIVError;
		tyP0940CommCtrl.tySOT.tyBtnAIVRdy3.bValue		:= p_tyDI.bSOT3AIVReady;
		tyP0940CommCtrl.tySOT.tyBtnAIVAvail3.bValue		:= p_tyDI.bSOT3AIVAvailable;
		tyP0940CommCtrl.tySOT.tyBtnAIVSLarge3.bValue	:= p_tyDI.bSOT3AIVSizeLarge;

		tyP0940CommCtrl.tySOT.tyBtnAIVRcv4.bValue		:= p_tyDI.bSOT4Receive;
		tyP0940CommCtrl.tySOT.tyBtnAIVErr4.bValue		:= p_tyDI.bSOT4AIVError;
		tyP0940CommCtrl.tySOT.tyBtnAIVRdy4.bValue		:= p_tyDI.bSOT4AIVReady;
		tyP0940CommCtrl.tySOT.tyBtnAIVAvail4.bValue		:= p_tyDI.bSOT4AIVAvailable;
		tyP0940CommCtrl.tySOT.tyBtnAIVSLarge4.bValue	:= p_tyDI.bSOT4AIVSizeLarge;

		tyP0940CommCtrl.tySOT.tyBtnFleetMgrActive.bValue := p_tyDI.bFleetManagerReady;

	ELSIF p_tyMcParamCurr.eAGVComProtocol = McSetAGVCommOPCUA AND p_tyNtParamCurr.bProjSOTSensorPrep = FALSE THEN

		tyP0940CommCtrl.tySOT.tyBtnAIVErr1.bValue		:= p_tyTagFromMes.tyTagStatOfPlatforms[1].bError;
		tyP0940CommCtrl.tySOT.tyBtnAIVRdy1.bValue		:= p_tyTagFromMes.tyTagStatOfPlatforms[1].bReady;
		tyP0940CommCtrl.tySOT.tyBtnAIVAvail1.bValue		:= p_tyTagFromMes.tyTagStatOfPlatforms[1].bAvailable;
		tyP0940CommCtrl.tySOT.tyBtnAIVSLarge1.bValue	:= p_tyTagFromMes.tyTagStatOfPlatforms[1].bSizeLarge;

		tyP0940CommCtrl.tySOT.tyBtnAIVErr2.bValue		:= p_tyTagFromMes.tyTagStatOfPlatforms[2].bError;
		tyP0940CommCtrl.tySOT.tyBtnAIVRdy2.bValue		:= p_tyTagFromMes.tyTagStatOfPlatforms[2].bReady;
		tyP0940CommCtrl.tySOT.tyBtnAIVAvail2.bValue		:= p_tyTagFromMes.tyTagStatOfPlatforms[2].bAvailable;
		tyP0940CommCtrl.tySOT.tyBtnAIVSLarge2.bValue	:= p_tyTagFromMes.tyTagStatOfPlatforms[2].bSizeLarge;

		tyP0940CommCtrl.tySOT.tyBtnAIVErr3.bValue		:= p_tyTagFromMes.tyTagStatOfPlatforms[3].bError;
		tyP0940CommCtrl.tySOT.tyBtnAIVRdy3.bValue		:= p_tyTagFromMes.tyTagStatOfPlatforms[3].bReady;
		tyP0940CommCtrl.tySOT.tyBtnAIVAvail3.bValue		:= p_tyTagFromMes.tyTagStatOfPlatforms[3].bAvailable;
		tyP0940CommCtrl.tySOT.tyBtnAIVSLarge3.bValue	:= p_tyTagFromMes.tyTagStatOfPlatforms[3].bSizeLarge;

		tyP0940CommCtrl.tySOT.tyBtnAIVErr4.bValue		:= p_tyTagFromMes.tyTagStatOfPlatforms[4].bError;
		tyP0940CommCtrl.tySOT.tyBtnAIVRdy4.bValue		:= p_tyTagFromMes.tyTagStatOfPlatforms[4].bReady;
		tyP0940CommCtrl.tySOT.tyBtnAIVAvail4.bValue		:= p_tyTagFromMes.tyTagStatOfPlatforms[4].bAvailable;
		tyP0940CommCtrl.tySOT.tyBtnAIVSLarge4.bValue	:= p_tyTagFromMes.tyTagStatOfPlatforms[4].bSizeLarge;

		tyP0940CommCtrl.tySOT.tyBtnFleetMgrActive.bValue := p_tyTagFromMes.bActive;
	END_IF

	IF p_tyMcParamCurr.eAGVComProtocol = McSetAGVCommDisabled THEN
		tyP0940CommCtrl.tySOT.tyBtnAIVErr1.bValue		:= FALSE;
		tyP0940CommCtrl.tySOT.tyBtnAIVRdy1.bValue		:= FALSE;
		tyP0940CommCtrl.tySOT.tyBtnAIVAvail1.bValue		:= FALSE;
		tyP0940CommCtrl.tySOT.tyBtnAIVSLarge1.bValue	:= FALSE;

		tyP0940CommCtrl.tySOT.tyBtnAIVErr2.bValue		:= FALSE;
		tyP0940CommCtrl.tySOT.tyBtnAIVRdy2.bValue		:= FALSE;
		tyP0940CommCtrl.tySOT.tyBtnAIVAvail2.bValue		:= FALSE;
		tyP0940CommCtrl.tySOT.tyBtnAIVSLarge2.bValue	:= FALSE;

		tyP0940CommCtrl.tySOT.tyBtnAIVErr3.bValue		:= FALSE;
		tyP0940CommCtrl.tySOT.tyBtnAIVRdy3.bValue		:= FALSE;
		tyP0940CommCtrl.tySOT.tyBtnAIVAvail3.bValue		:= FALSE;
		tyP0940CommCtrl.tySOT.tyBtnAIVSLarge3.bValue	:= FALSE;

		tyP0940CommCtrl.tySOT.tyBtnAIVErr4.bValue		:= FALSE;
		tyP0940CommCtrl.tySOT.tyBtnAIVRdy4.bValue		:= FALSE;
		tyP0940CommCtrl.tySOT.tyBtnAIVAvail4.bValue		:= FALSE;
		tyP0940CommCtrl.tySOT.tyBtnAIVSLarge4.bValue	:= FALSE;

		tyP0940CommCtrl.tySOT.tyBtnFleetMgrActive.bValue := FALSE;
	END_IF

	IF tyP0940CommCtrl.tyDMCRFID.tyLyr.uiRtStat.0 = 0  THEN //if hidden update
		tyP0940CommCtrl.tyDMCRFID.tyBtnScanComplSig.bValue		:= p_bDIPCBScanComplSig;

	END_IF
END_ACTION
```

#### Act_OptP0940WriteDO.st
```iecst
ACTION Act_OptP0940WriteDO:

	//USBA
	IF tyP0940CommCtrl.tyUSSMEMAA.tyBtnUSB.bRtCompl = TRUE THEN

		IF tyP0940CommCtrl.tyUSSMEMAA.tyBtnUSB.bValue = TRUE THEN
			eUSSMEMAAAct	:= SMEMAActSetSig;

			IF p_eUSSMEMAAStat = SMEMAActSetSig AND p_eUSSMEMAAStatus = Done THEN
				eUSSMEMAAAct	:= SMEMAActIdle;

				tyP0940CommCtrl.tyUSSMEMAA.tyBtnUSB.bRtCompl	:= FALSE;
			END_IF

		ELSE
			eUSSMEMAAAct	:= SMEMAActRstSig;

			IF p_eUSSMEMAAStat = SMEMAActRstSig AND p_eUSSMEMAAStatus = Done THEN
				eUSSMEMAAAct	:= SMEMAActIdle;

				tyP0940CommCtrl.tyUSSMEMAA.tyBtnUSB.bRtCompl	:= FALSE;
			END_IF

		END_IF

	END_IF

	//USBB
	IF tyP0940CommCtrl.tyUSSMEMAB.tyBtnUSB.bRtCompl = TRUE THEN

		IF tyP0940CommCtrl.tyUSSMEMAB.tyBtnUSB.bValue = TRUE THEN
			eUSSMEMABAct	:= SMEMAActSetSig;

			IF p_eUSSMEMABStat = SMEMAActSetSig AND p_eUSSMEMABStatus = Done THEN
				eUSSMEMABAct	:= SMEMAActIdle;

				tyP0940CommCtrl.tyUSSMEMAB.tyBtnUSB.bRtCompl	:= FALSE;
			END_IF

		ELSE
			eUSSMEMABAct	:= SMEMAActRstSig;

			IF p_eUSSMEMABStat = SMEMAActRstSig AND p_eUSSMEMABStatus = Done THEN
				eUSSMEMABAct	:= SMEMAActIdle;

				tyP0940CommCtrl.tyUSSMEMAB.tyBtnUSB.bRtCompl	:= FALSE;
			END_IF

		END_IF

	END_IF

	IF p_tyMcParamCurr.eAGVComProtocol <> McSetAGVCommDisabled THEN
		//Error
		IF tyP0940CommCtrl.tySOT.tyBtnMagErr1.bRtCompl = TRUE THEN

			IF tyP0940CommCtrl.tySOT.tyBtnMagErr1.bValue = TRUE THEN
				bSOTMagErr1 := TRUE;
				tyP0940CommCtrl.tySOT.tyBtnMagErr1.bRtCompl := FALSE;
			ELSE
				bSOTMagErr1 := FALSE;
				tyP0940CommCtrl.tySOT.tyBtnMagErr1.bRtCompl := FALSE;
			END_IF
		END_IF

		IF tyP0940CommCtrl.tySOT.tyBtnMagErr2.bRtCompl = TRUE THEN

			IF tyP0940CommCtrl.tySOT.tyBtnMagErr2.bValue = TRUE THEN
				bSOTMagErr2 := TRUE;
				tyP0940CommCtrl.tySOT.tyBtnMagErr2.bRtCompl := FALSE;
			ELSE
				bSOTMagErr2 := FALSE;
				tyP0940CommCtrl.tySOT.tyBtnMagErr2.bRtCompl := FALSE;
			END_IF
		END_IF

		IF tyP0940CommCtrl.tySOT.tyBtnMagErr3.bRtCompl = TRUE THEN

			IF tyP0940CommCtrl.tySOT.tyBtnMagErr3.bValue = TRUE THEN
				bSOTMagErr3 := TRUE;
				tyP0940CommCtrl.tySOT.tyBtnMagErr3.bRtCompl := FALSE;
			ELSE
				bSOTMagErr3 := FALSE;
				tyP0940CommCtrl.tySOT.tyBtnMagErr3.bRtCompl := FALSE;
			END_IF
		END_IF

		IF tyP0940CommCtrl.tySOT.tyBtnMagErr4.bRtCompl = TRUE THEN

			IF tyP0940CommCtrl.tySOT.tyBtnMagErr4.bValue = TRUE THEN
				bSOTMagErr4 := TRUE;
				tyP0940CommCtrl.tySOT.tyBtnMagErr4.bRtCompl := FALSE;
			ELSE
				bSOTMagErr4 := FALSE;
				tyP0940CommCtrl.tySOT.tyBtnMagErr4.bRtCompl := FALSE;
			END_IF
		END_IF

		//Ready
		IF tyP0940CommCtrl.tySOT.tyBtnMagRdy1.bRtCompl = TRUE THEN

			IF tyP0940CommCtrl.tySOT.tyBtnMagRdy1.bValue = TRUE THEN
				bSOTMagRdy1 := TRUE;
				tyP0940CommCtrl.tySOT.tyBtnMagRdy1.bRtCompl := FALSE;
			ELSE
				bSOTMagRdy1 := FALSE;
				tyP0940CommCtrl.tySOT.tyBtnMagRdy1.bRtCompl := FALSE;
			END_IF
		END_IF

		IF tyP0940CommCtrl.tySOT.tyBtnMagRdy2.bRtCompl = TRUE THEN

			IF tyP0940CommCtrl.tySOT.tyBtnMagRdy2.bValue = TRUE THEN
				bSOTMagRdy2 := TRUE;
				tyP0940CommCtrl.tySOT.tyBtnMagRdy2.bRtCompl := FALSE;
			ELSE
				bSOTMagRdy2 := FALSE;
				tyP0940CommCtrl.tySOT.tyBtnMagRdy2.bRtCompl := FALSE;
			END_IF
		END_IF

		IF tyP0940CommCtrl.tySOT.tyBtnMagRdy3.bRtCompl = TRUE THEN

			IF tyP0940CommCtrl.tySOT.tyBtnMagRdy3.bValue = TRUE THEN
				bSOTMagRdy3 := TRUE;
				tyP0940CommCtrl.tySOT.tyBtnMagRdy3.bRtCompl := FALSE;
			ELSE
				bSOTMagRdy3 := FALSE;
				tyP0940CommCtrl.tySOT.tyBtnMagRdy3.bRtCompl := FALSE;
			END_IF
		END_IF

		IF tyP0940CommCtrl.tySOT.tyBtnMagRdy4.bRtCompl = TRUE THEN

			IF tyP0940CommCtrl.tySOT.tyBtnMagRdy4.bValue = TRUE THEN
				bSOTMagRdy4 := TRUE;
				tyP0940CommCtrl.tySOT.tyBtnMagRdy4.bRtCompl := FALSE;
			ELSE
				bSOTMagRdy4 := FALSE;
				tyP0940CommCtrl.tySOT.tyBtnMagRdy4.bRtCompl := FALSE;
			END_IF
		END_IF

		//Available
		IF tyP0940CommCtrl.tySOT.tyBtnMagAvail1.bRtCompl = TRUE THEN

			IF tyP0940CommCtrl.tySOT.tyBtnMagAvail1.bValue = TRUE THEN
				bSOTMagAvail1 := TRUE;
				tyP0940CommCtrl.tySOT.tyBtnMagAvail1.bRtCompl := FALSE;
			ELSE
				bSOTMagAvail1 := FALSE;
				tyP0940CommCtrl.tySOT.tyBtnMagAvail1.bRtCompl := FALSE;
			END_IF
		END_IF

		IF tyP0940CommCtrl.tySOT.tyBtnMagAvail2.bRtCompl = TRUE THEN

			IF tyP0940CommCtrl.tySOT.tyBtnMagAvail2.bValue = TRUE THEN
				bSOTMagAvail2 := TRUE;
				tyP0940CommCtrl.tySOT.tyBtnMagAvail2.bRtCompl := FALSE;
			ELSE
				bSOTMagAvail2 := FALSE;
				tyP0940CommCtrl.tySOT.tyBtnMagAvail2.bRtCompl := FALSE;
			END_IF
		END_IF

		IF tyP0940CommCtrl.tySOT.tyBtnMagAvail3.bRtCompl = TRUE THEN

			IF tyP0940CommCtrl.tySOT.tyBtnMagAvail3.bValue = TRUE THEN
				bSOTMagAvail3 := TRUE;
				tyP0940CommCtrl.tySOT.tyBtnMagAvail3.bRtCompl := FALSE;
			ELSE
				bSOTMagAvail3 := FALSE;
				tyP0940CommCtrl.tySOT.tyBtnMagAvail3.bRtCompl := FALSE;
			END_IF
		END_IF

		IF tyP0940CommCtrl.tySOT.tyBtnMagAvail4.bRtCompl = TRUE THEN

			IF tyP0940CommCtrl.tySOT.tyBtnMagAvail4.bValue = TRUE THEN
				bSOTMagAvail4 := TRUE;
				tyP0940CommCtrl.tySOT.tyBtnMagAvail4.bRtCompl := FALSE;
			ELSE
				bSOTMagAvail4 := FALSE;
				tyP0940CommCtrl.tySOT.tyBtnMagAvail4.bRtCompl := FALSE;
			END_IF
		END_IF

		//Size
		IF tyP0940CommCtrl.tySOT.tyBtnMagSLarge1.bRtCompl = TRUE THEN

			IF tyP0940CommCtrl.tySOT.tyBtnMagSLarge1.bValue = TRUE THEN
				bSOTMagSLarge1 := TRUE;
				tyP0940CommCtrl.tySOT.tyBtnMagSLarge1.bRtCompl := FALSE;
			ELSE
				bSOTMagSLarge1 := FALSE;
				tyP0940CommCtrl.tySOT.tyBtnMagSLarge1.bRtCompl := FALSE;
			END_IF
		END_IF

		IF tyP0940CommCtrl.tySOT.tyBtnMagSLarge2.bRtCompl = TRUE THEN

			IF tyP0940CommCtrl.tySOT.tyBtnMagSLarge2.bValue = TRUE THEN
				bSOTMagSLarge2 := TRUE;
				tyP0940CommCtrl.tySOT.tyBtnMagSLarge2.bRtCompl := FALSE;
			ELSE
				bSOTMagSLarge2 := FALSE;
				tyP0940CommCtrl.tySOT.tyBtnMagSLarge2.bRtCompl := FALSE;
			END_IF
		END_IF

		IF tyP0940CommCtrl.tySOT.tyBtnMagSLarge3.bRtCompl = TRUE THEN

			IF tyP0940CommCtrl.tySOT.tyBtnMagSLarge3.bValue = TRUE THEN
				bSOTMagSLarge3 := TRUE;
				tyP0940CommCtrl.tySOT.tyBtnMagSLarge3.bRtCompl := FALSE;
			ELSE
				bSOTMagSLarge3 := FALSE;
				tyP0940CommCtrl.tySOT.tyBtnMagSLarge3.bRtCompl := FALSE;
			END_IF
		END_IF

		IF tyP0940CommCtrl.tySOT.tyBtnMagSLarge4.bRtCompl = TRUE THEN

			IF tyP0940CommCtrl.tySOT.tyBtnMagSLarge4.bValue = TRUE THEN
				bSOTMagSLarge4 := TRUE;
				tyP0940CommCtrl.tySOT.tyBtnMagSLarge4.bRtCompl := FALSE;
			ELSE
				bSOTMagSLarge4 := FALSE;
				tyP0940CommCtrl.tySOT.tyBtnMagSLarge4.bRtCompl := FALSE;
			END_IF
		END_IF

		//Req Bring
		IF tyP0940CommCtrl.tySOT.tyBtnMagReqBring1.bRtCompl = TRUE THEN

			IF tyP0940CommCtrl.tySOT.tyBtnMagReqBring1.bValue = TRUE THEN
				bAIVReqBring1 := TRUE;
				tyP0940CommCtrl.tySOT.tyBtnMagReqBring1.bRtCompl := FALSE;
			ELSE
				bAIVReqBring1 := FALSE;
				tyP0940CommCtrl.tySOT.tyBtnMagReqBring1.bRtCompl := FALSE;
			END_IF
		END_IF

		IF tyP0940CommCtrl.tySOT.tyBtnMagReqBring2.bRtCompl = TRUE THEN

			IF tyP0940CommCtrl.tySOT.tyBtnMagReqBring2.bValue = TRUE THEN
				bAIVReqBring2 := TRUE;
				tyP0940CommCtrl.tySOT.tyBtnMagReqBring2.bRtCompl := FALSE;
			ELSE
				bAIVReqBring2 := FALSE;
				tyP0940CommCtrl.tySOT.tyBtnMagReqBring2.bRtCompl := FALSE;
			END_IF
		END_IF

		IF tyP0940CommCtrl.tySOT.tyBtnMagReqBring3.bRtCompl = TRUE THEN

			IF tyP0940CommCtrl.tySOT.tyBtnMagReqBring3.bValue = TRUE THEN
				bAIVReqBring1 := TRUE;
				tyP0940CommCtrl.tySOT.tyBtnMagReqBring3.bRtCompl := FALSE;
			ELSE
				bAIVReqBring1 := FALSE;
				tyP0940CommCtrl.tySOT.tyBtnMagReqBring3.bRtCompl := FALSE;
			END_IF
		END_IF

		IF tyP0940CommCtrl.tySOT.tyBtnMagReqBring4.bRtCompl = TRUE THEN

			IF tyP0940CommCtrl.tySOT.tyBtnMagReqBring4.bValue = TRUE THEN
				bAIVReqBring1 := TRUE;
				tyP0940CommCtrl.tySOT.tyBtnMagReqBring4.bRtCompl := FALSE;
			ELSE
				bAIVReqBring1 := FALSE;
				tyP0940CommCtrl.tySOT.tyBtnMagReqBring4.bRtCompl := FALSE;
			END_IF
		END_IF

		//Req Get
		IF tyP0940CommCtrl.tySOT.tyBtnMagReqtGet1.bRtCompl = TRUE THEN

			IF tyP0940CommCtrl.tySOT.tyBtnMagReqtGet1.bValue = TRUE THEN
				bAIVReqGet1 := TRUE;
				tyP0940CommCtrl.tySOT.tyBtnMagReqtGet1.bRtCompl := FALSE;
			ELSE
				bAIVReqGet1 := FALSE;
				tyP0940CommCtrl.tySOT.tyBtnMagReqtGet1.bRtCompl := FALSE;
			END_IF
		END_IF

		IF tyP0940CommCtrl.tySOT.tyBtnMagReqtGet2.bRtCompl = TRUE THEN

			IF tyP0940CommCtrl.tySOT.tyBtnMagReqtGet2.bValue = TRUE THEN
				bAIVReqGet2 := TRUE;
				tyP0940CommCtrl.tySOT.tyBtnMagReqtGet2.bRtCompl := FALSE;
			ELSE
				bAIVReqGet2 := FALSE;
				tyP0940CommCtrl.tySOT.tyBtnMagReqtGet2.bRtCompl := FALSE;
			END_IF
		END_IF

		IF tyP0940CommCtrl.tySOT.tyBtnMagReqtGet3.bRtCompl = TRUE THEN

			IF tyP0940CommCtrl.tySOT.tyBtnMagReqtGet3.bValue = TRUE THEN
				bAIVReqGet3 := TRUE;
				tyP0940CommCtrl.tySOT.tyBtnMagReqtGet3.bRtCompl := FALSE;
			ELSE
				bAIVReqGet3 := FALSE;
				tyP0940CommCtrl.tySOT.tyBtnMagReqtGet3.bRtCompl := FALSE;
			END_IF
		END_IF

		IF tyP0940CommCtrl.tySOT.tyBtnMagReqtGet4.bRtCompl = TRUE THEN

			IF tyP0940CommCtrl.tySOT.tyBtnMagReqtGet4.bValue = TRUE THEN
				bAIVReqGet4 := TRUE;
				tyP0940CommCtrl.tySOT.tyBtnMagReqtGet4.bRtCompl := FALSE;
			ELSE
				bAIVReqGet4 := FALSE;
				tyP0940CommCtrl.tySOT.tyBtnMagReqtGet4.bRtCompl := FALSE;
			END_IF
		END_IF
	END_IF

	//DMC Start Scan
	IF tyP0940CommCtrl.tyDMCRFID.tyLyr.uiRtStat.0 = 0 THEN
		IF tyP0940CommCtrl.tyDMCRFID.tyBtnTrigStartScan.bRtCompl = TRUE THEN
			IF tyP0940CommCtrl.tyDMCRFID.tyBtnTrigStartScan.bValue = TRUE THEN
				bStartScanSig := TRUE;
			ELSE
				bStartScanSig := FALSE;
			END_IF
		END_IF
		IF tyP0940CommCtrl.tyDMCRFID.tyBtnTrigTransMag1Out.bRtCompl = TRUE THEN
			IF tyP0940CommCtrl.tyDMCRFID.tyBtnTrigTransMag1Out.bValue = TRUE THEN
				bPCBExitMag1 := TRUE;
			ELSE
				bPCBExitMag1 := FALSE;
			END_IF
		END_IF
		IF tyP0940CommCtrl.tyDMCRFID.tyBtnTrigTransMag2Out.bRtCompl = TRUE THEN
			IF tyP0940CommCtrl.tyDMCRFID.tyBtnTrigTransMag2Out.bValue = TRUE THEN
				bPCBExitMag2 := TRUE;
			ELSE
				bPCBExitMag2 := FALSE;
			END_IF
		END_IF
		IF tyP0940CommCtrl.tyDMCRFID.tyBtnTrigTransMag3Out.bRtCompl = TRUE THEN
			IF tyP0940CommCtrl.tyDMCRFID.tyBtnTrigTransMag3Out.bValue = TRUE THEN
				bPCBExitMag3 := TRUE;
			ELSE
				bPCBExitMag3 := FALSE;
			END_IF
		END_IF
	END_IF
END_ACTION
```

#### Act_OptP0940RstMnl.st
```iecst
ACTION Act_OptP0940RstMnl:

	IF EDGEPOS((bManualMod = FALSE) OR (p_eUSSMEMAAStatus = Error)) THEN
		eUSSMEMAAAct	:= SMEMAActIdle;

		tyP0940CommCtrl.tyUSSMEMAA.tyBtnUSB.bValue	:= FALSE;
	END_IF

	IF EDGEPOS((bManualMod = FALSE) OR (p_eUSSMEMABStatus = Error)) THEN
		eUSSMEMABAct	:= SMEMAActIdle;

		tyP0940CommCtrl.tyUSSMEMAB.tyBtnUSB.bValue	:= FALSE;
	END_IF

	IF EDGEPOS(bManualMod = FALSE) THEN
		tyP0940CommCtrl.tySOT.tyBtnMagErr1.bValue := FALSE;
		tyP0940CommCtrl.tySOT.tyBtnMagErr2.bValue := FALSE;
		tyP0940CommCtrl.tySOT.tyBtnMagErr3.bValue := FALSE;
		tyP0940CommCtrl.tySOT.tyBtnMagErr4.bValue := FALSE;

		tyP0940CommCtrl.tySOT.tyBtnMagRdy1.bValue := FALSE;
		tyP0940CommCtrl.tySOT.tyBtnMagRdy2.bValue := FALSE;
		tyP0940CommCtrl.tySOT.tyBtnMagRdy3.bValue := FALSE;
		tyP0940CommCtrl.tySOT.tyBtnMagRdy4.bValue := FALSE;

		tyP0940CommCtrl.tySOT.tyBtnMagAvail1.bValue := FALSE;
		tyP0940CommCtrl.tySOT.tyBtnMagAvail2.bValue := FALSE;
		tyP0940CommCtrl.tySOT.tyBtnMagAvail3.bValue := FALSE;
		tyP0940CommCtrl.tySOT.tyBtnMagAvail4.bValue := FALSE;

		tyP0940CommCtrl.tySOT.tyBtnMagSLarge1.bValue := FALSE;
		tyP0940CommCtrl.tySOT.tyBtnMagSLarge2.bValue := FALSE;
		tyP0940CommCtrl.tySOT.tyBtnMagSLarge3.bValue := FALSE;
		tyP0940CommCtrl.tySOT.tyBtnMagSLarge4.bValue := FALSE;

		bSOTMagErr1 := FALSE;
		bSOTMagErr2 := FALSE;
		bSOTMagErr3 := FALSE;
		bSOTMagErr4 := FALSE;

		bSOTMagRdy1 := FALSE;
		bSOTMagRdy2 := FALSE;
		bSOTMagRdy3 := FALSE;
		bSOTMagRdy4 := FALSE;

		bSOTMagAvail1 := FALSE;
		bSOTMagAvail2 := FALSE;
		bSOTMagAvail3 := FALSE;
		bSOTMagAvail4 := FALSE;

		bSOTMagSLarge1 := FALSE;
		bSOTMagSLarge2 := FALSE;
		bSOTMagSLarge3 := FALSE;
		bSOTMagSLarge4 := FALSE;

		bAIVReqBring1 := FALSE;
		bAIVReqBring2 := FALSE;
		bAIVReqBring3 := FALSE;
		bAIVReqBring4 := FALSE;

		bAIVReqGet1 := FALSE;
		bAIVReqGet2 := FALSE;
		bAIVReqGet3 := FALSE;
		bAIVReqGet4 := FALSE;

		bStartScanSig := FALSE;
		bPCBExitMag1 := FALSE;
		bPCBExitMag2 := FALSE;
		bPCBExitMag3 := FALSE;
	END_IF

END_ACTION
```

#### Act_EntP0950Disp.st
```iecst
ACTION Act_EntP0950Disp:

	// Access Address
	p_tyC0002FullMask ACCESS ADR (tyP0950Simu.tyFullMaskHide);

	p_tyC0005Main ACCESS ADR(tyCommon.tyMain);

	p_tyC0007Notif ACCESS ADR(tyCommon.tyNotif);

	p_tyC0009Info ACCESS ADR(tyCommon.tyInfo);

	p_tyP0950Simu ACCESS ADR(tyP0950Simu.tySimu);

	p_tyP0950SimuCycleTim ACCESS ADR(tyP0950Simu.tySimuBffrCycleTm);

	p_tyP0950SimuAGVtoMC ACCESS ADR(tyP0950Simu.tyAGVToMc);

	p_tyP0950SimuMCtoAGV ACCESS ADR(tyP0950Simu.tyMcToAGV);

	//Display

	tyP0950Simu.tySimu.tyNumTravSpd.diValue := p_diNtParamTravAutoSpd;
	tyP0950Simu.tySimu.tyNumLifterSpd.diValue := p_diNtParamLifterAutoSpd;
	tyP0950Simu.tySimu.tyNumAddr.diValue := p_usiNtParamNtAddr;
	tyP0950Simu.tySimu.tyStringJobNo.sValue:= p_sNtParamJobNo;
END_ACTION
```

#### Act_OptP0950Navi.st
```iecst
ACTION Act_OptP0950Navi:

	IF tyP0950Simu.tySimu.tyBtnNavLeft.bRtCompl OR tyP0950Simu.tySimu.tyBtnNavRight.bRtCompl THEN
		tyP0950Simu.tyAGVToMc.tyBtnNavLeft.bRtCompl := FALSE;
		tyP0950Simu.tySimu.tyBtnNavRight.bRtCompl := FALSE;

		fUIInRtStatHide(ADR(tyP0950Simu.tyAGVToMc.tyLyr.uiRtStat));
		fUIInRtStatHide(ADR(tyP0950Simu.tySimu.tyLyr1.uiRtStat));
		fUIInRtStatHide(ADR(tyP0950Simu.tySimu.tyLyr2.uiRtStat));
		fUIInRtStatOff(ADR(tyP0950Simu.tySimuBffrCycleTm.tyLyr.uiRtStat));
	ELSIF tyP0950Simu.tySimuBffrCycleTm.tyBtnNavRight.bRtCompl OR tyP0950Simu.tySimuBffrCycleTm.tyBtnNavLeft.bRtCompl THEN
		tyP0950Simu.tyAGVToMc.tyBtnNavRight.bRtCompl  := FALSE;
		tyP0950Simu.tySimuBffrCycleTm.tyBtnNavLeft.bRtCompl  := FALSE;

		fUIInRtStatHide(ADR(tyP0950Simu.tyAGVToMc.tyLyr.uiRtStat));
		fUIInRtStatHide(ADR(tyP0950Simu.tySimuBffrCycleTm.tyLyr.uiRtStat));
		fUIInRtStatOff(ADR(tyP0950Simu.tySimu.tyLyr1.uiRtStat));
		fUIInRtStatOff(ADR(tyP0950Simu.tySimu.tyLyr2.uiRtStat));
//	ELSIF tyP0950Simu.tySimuBffrCycleTm.tyBtnNavRight.bRtCompl OR tyP0950Simu.tySimu.tyBtnNavLeft.bRtCompl THEN
//		tyP0950Simu.tySimuBffrCycleTm.tyBtnNavRight.bRtCompl  := FALSE;
//		tyP0950Simu.tySimu.tyBtnNavLeft.bRtCompl  := FALSE;
//
//		fUIInRtStatHide(ADR(tyP0950Simu.tySimu.tyLyr1.uiRtStat));
//		fUIInRtStatHide(ADR(tyP0950Simu.tySimu.tyLyr2.uiRtStat));
//		fUIInRtStatHide(ADR(tyP0950Simu.tySimuBffrCycleTm.tyLyr.uiRtStat));
//		fUIInRtStatOff(ADR(tyP0950Simu.tyAGVToMc.tyLyr.uiRtStat));
	END_IF

END_ACTION
```

#### Act_OptP0950SimuMod.st
```iecst
ACTION Act_OptP0950SimuMod:

//	IF EDGEPOS(tyOpsProgData.bSimuCtrl) THEN
//		g_tyP0950Simu.tySimu.tyBtnEngageTest.bRtLk		:= TRUE;
//	ELSIF EDGENEG(tyOpsProgData.bSimuCtrl) THEN
//		g_tyP0950Simu.tySimu.tyBtnEngageTest.bRtLk		:= g_tyP0950Simu.tySimu.tyBtnEngageTest.bValue;
//	END_IF
//
//	IF g_tyP0950Simu.tySimu.tyBtnEngageTest.bRtCompl THEN
//		g_tyP0950Simu.tySimu.tyBtnEngageTest.bRtCompl 	:= FALSE;
//		g_tyP0950Simu.tySimu.tyBtnEngageTest.bValue	  	:= TRUE;
//		g_tyP0950Simu.tySimu.tyBtnEngageTest.bRtLk	  	:= TRUE;
//
//		usiSimuMod				:= 0;
//	END_IF

	IF p_bSimuStatusRun THEN
		tyP0950Simu.tySimu.tyBtnSimu.bRtLk				:= TRUE;
	ELSE
		tyP0950Simu.tySimu.tyBtnSimu.bRtLk				:= tyP0950Simu.tySimu.tyBtnSimu.bValue;
	END_IF

	IF tyP0950Simu.tySimu.tyBtnSimu.bRtCompl THEN
		tyP0950Simu.tySimu.tyBtnSimu.bRtCompl 			:= FALSE;
		tyP0950Simu.tySimu.tyBtnSimu.bValue	  			:= TRUE;
		tyP0950Simu.tySimu.tyBtnSimu.bRtLk	  			:= TRUE;
	END_IF

END_ACTION
```

#### Act_OptP0950Ctrl.st
```iecst
ACTION Act_OptP0950Ctrl:

	// Error
	IF EDGEPOS(p_bAlarmErr = TRUE AND p_bSimuStatusStop = FALSE) THEN

		tyP0950Simu.tySimu.tyBtnStart.bRtCompl	:= FALSE;
		tyP0950Simu.tySimu.tyBtnStop.bRtCompl	:= FALSE;

		tyP0950Simu.tySimu.tyBtnStart.bValue	:= FALSE;
		tyP0950Simu.tySimu.tyBtnStop.bValue		:= FALSE;

		eSimuAct	:= SimulationsActError;
		bAGVSimulationOn	:= FALSE;
	ELSE

		IF p_eSimuStat = SimulationsActError AND p_eSimuStatus = Done THEN
			eSimuAct	:= SimulationsActIdle;
			bAGVSimulationOn	:= FALSE;
		END_IF

	END_IF

	//Control
	IF tyP0950Simu.tySimu.tyBtnStart.bRtCompl = TRUE THEN
		tyP0950Simu.tySimu.tyBtnStop.bRtCompl	:= FALSE;
		bAGVSimulationOn	:= TRUE;
		eSimuAct		:= SimulationsActStart;

		IF p_eSimuStat = SimulationsActStart AND p_eSimuStatus = Done THEN
			eSimuAct	:= SimulationsActIdle;

			tyP0950Simu.tySimu.tyBtnStart.bRtCompl	:= FALSE;

		END_IF

	ELSIF tyP0950Simu.tySimu.tyBtnStop.bRtCompl = TRUE THEN
		tyP0950Simu.tySimu.tyBtnStart.bRtCompl	:= FALSE;
		bAGVSimulationOn	:= FALSE;
		eSimuAct			:= SimulationsActStop;

		IF p_eSimuStat = SimulationsActStop AND p_eSimuStatus = Done THEN
			eSimuAct		:= SimulationsActIdle;

			tyP0950Simu.tySimu.tyBtnStart.bValue	:= FALSE;
			tyP0950Simu.tySimu.tyBtnStop.bRtCompl	:= FALSE;
		END_IF

	END_IF

	// Mask
	IF p_bAlarmErr = TRUE OR (p_tyDI.bSafetyRlySig = FALSE) THEN
		fUIInRtStatOff(ADR(tyP0950Simu.tySimu.tyBtnStart.uiMaskRtStat));
		fUIInRtStatOff(ADR(tyP0950Simu.tySimu.tyBtnStop.uiMaskRtStat));
		tyP0950Simu.tySimu.tyBtnStart.bValue	:= FALSE;
		bAGVSimulationOn	:= FALSE;
	ELSIF p_bSimuStatusCycleStop = TRUE THEN
		fUIInRtStatHide(ADR(tyP0950Simu.tySimu.tyBtnStart.uiMaskRtStat));
		fUIInRtStatOff(ADR(tyP0950Simu.tySimu.tyBtnStop.uiMaskRtStat));
		tyP0950Simu.tySimu.tyBtnStart.bValue	:= FALSE;
		bAGVSimulationOn	:= FALSE;
		fbStopBlinkTm(IN := TRUE);
		IF fbStopBlinkTm.Q = TRUE THEN
			fbStopBlinkTm(IN := FALSE);

			tyP0950Simu.tySimu.tyBtnStart.bValue		:= NOT tyP0950Simu.tySimu.tyBtnStart.bValue;
		END_IF

	ELSIF p_bSimuStatusRun = TRUE THEN
		fUIInRtStatOff(ADR(tyP0950Simu.tySimu.tyBtnStart.uiMaskRtStat));
		fUIInRtStatHide(ADR(tyP0950Simu.tySimu.tyBtnStop.uiMaskRtStat));

	ELSE
		fUIInRtStatHide(ADR(tyP0950Simu.tySimu.tyBtnStart.uiMaskRtStat));
		fUIInRtStatOff(ADR(tyP0950Simu.tySimu.tyBtnStop.uiMaskRtStat));

	END_IF

	//AGV Simulatiom
	IF tyP0950Simu.tyAGVToMc.tyBtnAGVSimulateOn.bRtCompl THEN
		IF tyP0950Simu.tyAGVToMc.tyBtnAGVSimulateOn.bValue THEN
			bAGVSimulationOn	:= TRUE;
			tyP0950Simu.tyAGVToMc.tyBtnAGVSimulateOn.bRtCompl:= FALSE;
		ELSE
			bAGVSimulationOn := FALSE;
			tyP0950Simu.tyAGVToMc.tyBtnAGVSimulateOn.bRtCompl:= FALSE;
		END_IF
	END_IF

	IF tyP0950Simu.tyAGVToMc.tyBtnAGVOnline.bRtCompl THEN
		IF tyP0950Simu.tyAGVToMc.tyBtnAGVOnline.bValue THEN
			bAGVSimulateOnline := TRUE;
			tyP0950Simu.tyAGVToMc.tyBtnAGVOnline.bRtCompl := FALSE;
		ELSE
			bAGVSimulateOnline := FALSE;
			tyP0950Simu.tyAGVToMc.tyBtnAGVOnline.bRtCompl := FALSE;
		END_IF
	END_IF

	IF tyP0950Simu.tyAGVToMc.tyBtnAGVAuto.bRtCompl THEN
		IF tyP0950Simu.tyAGVToMc.tyBtnAGVAuto.bValue THEN
			tyAGVSimulateSig.bVEHAuto := TRUE;
			tyP0950Simu.tyAGVToMc.tyBtnAGVAuto.bRtCompl:= FALSE;
		ELSE
			tyAGVSimulateSig.bVEHAuto := FALSE;
			tyP0950Simu.tyAGVToMc.tyBtnAGVAuto.bRtCompl:= FALSE;
		END_IF
	END_IF

	IF tyP0950Simu.tyAGVToMc.tyBtnAGVInPos1.bRtCompl THEN
		IF tyP0950Simu.tyAGVToMc.tyBtnAGVInPos1.bValue THEN
			tyAGVSimulateSig.bVEHInPos1 := TRUE;
			tyP0950Simu.tyAGVToMc.tyBtnAGVInPos1.bRtCompl:= FALSE;
		ELSE
			tyAGVSimulateSig.bVEHInPos1 := FALSE;
			tyP0950Simu.tyAGVToMc.tyBtnAGVInPos1.bRtCompl:= FALSE;
		END_IF
	END_IF

	IF tyP0950Simu.tyAGVToMc.tyBtnAGVInPos2.bRtCompl THEN
		IF tyP0950Simu.tyAGVToMc.tyBtnAGVInPos2.bValue THEN
			tyAGVSimulateSig.bVEHInPos2 := TRUE;
			tyP0950Simu.tyAGVToMc.tyBtnAGVInPos2.bRtCompl:= FALSE;
		ELSE
			tyAGVSimulateSig.bVEHInPos2 := FALSE;
			tyP0950Simu.tyAGVToMc.tyBtnAGVInPos2.bRtCompl:= FALSE;
		END_IF
	END_IF

	IF tyP0950Simu.tyAGVToMc.tyBtnAGVInPos3.bRtCompl THEN
		IF tyP0950Simu.tyAGVToMc.tyBtnAGVInPos3.bValue THEN
			tyAGVSimulateSig.bVEHInPos3 := TRUE;
			tyP0950Simu.tyAGVToMc.tyBtnAGVInPos3.bRtCompl:= FALSE;
		ELSE
			tyAGVSimulateSig.bVEHInPos3 := FALSE;
			tyP0950Simu.tyAGVToMc.tyBtnAGVInPos3.bRtCompl:= FALSE;
		END_IF
	END_IF

	IF tyP0950Simu.tyAGVToMc.tyBtnAGV1Occupied.bRtCompl THEN
		IF tyP0950Simu.tyAGVToMc.tyBtnAGV1Occupied.bValue THEN
			tyAGVSimulateSig.bVEH1Occupied := TRUE;
			tyP0950Simu.tyAGVToMc.tyBtnAGV1Occupied.bRtCompl := FALSE;
		ELSE
			tyAGVSimulateSig.bVEH1Occupied := FALSE;
			tyP0950Simu.tyAGVToMc.tyBtnAGV1Occupied.bRtCompl := FALSE;
		END_IF
	END_IF

	IF tyP0950Simu.tyAGVToMc.tyBtnAGV2Occupied.bRtCompl THEN
		IF tyP0950Simu.tyAGVToMc.tyBtnAGV2Occupied.bValue THEN
			tyAGVSimulateSig.bVEH2Occupied := TRUE;
			tyP0950Simu.tyAGVToMc.tyBtnAGV2Occupied.bRtCompl := FALSE;
		ELSE
			tyAGVSimulateSig.bVEH2Occupied := FALSE;
			tyP0950Simu.tyAGVToMc.tyBtnAGV2Occupied.bRtCompl := FALSE;
		END_IF
	END_IF

	IF tyP0950Simu.tyAGVToMc.tyBtnAGV3Occupied.bRtCompl THEN
		IF tyP0950Simu.tyAGVToMc.tyBtnAGV3Occupied.bValue THEN
			tyAGVSimulateSig.bVEH3Occupied := TRUE;
			tyP0950Simu.tyAGVToMc.tyBtnAGV3Occupied.bRtCompl := FALSE;
		ELSE
			tyAGVSimulateSig.bVEH3Occupied := FALSE;
			tyP0950Simu.tyAGVToMc.tyBtnAGV3Occupied.bRtCompl := FALSE;
		END_IF
	END_IF

	//Machine to AGV Communication
	tyP0950Simu.tyMcToAGV.tyBtnMachineOnline.bValue := p_bMachineOnline;
	tyP0950Simu.tyMcToAGV.tyBtnMachineEstop.bValue	:= p_tyDTMagToAGV.bEStopErr;

	//Magazine #1 to AGV Communication
	tyP0950Simu.tyMcToAGV.tyBtnMag1Auto.bValue				:= p_tyDTMagToAGV.bCI1Auto;
	tyP0950Simu.tyMcToAGV.tyBtnMag1Empty.bValue				:= p_tyDTMagToAGV.bCI1MagazineFull;
	tyP0950Simu.tyMcToAGV.tyBtnMag1IncorrectModel.bValue	:= p_tyDTMagToAGV.bCI1IncorrectMagazineModel;
	tyP0950Simu.tyMcToAGV.tyBtnMag1Occupied.bValue			:= p_tyDTMagToAGV.bCI1Occupied;
	tyP0950Simu.tyMcToAGV.tyBtnMag1Rdy.bValue				:= p_tyDTMagToAGV.bCI1Rdy;

	//Magazine #2 to AGV Communication
	tyP0950Simu.tyMcToAGV.tyBtnMag2Auto.bValue				:= p_tyDTMagToAGV.bCI2Auto;
	tyP0950Simu.tyMcToAGV.tyBtnMag2Empty.bValue				:= p_tyDTMagToAGV.bCI2MagazineFull;
	tyP0950Simu.tyMcToAGV.tyBtnMag2IncorrectModel.bValue	:= p_tyDTMagToAGV.bCI2IncorrectMagazineModel;
	tyP0950Simu.tyMcToAGV.tyBtnMag2Occupied.bValue			:= p_tyDTMagToAGV.bCI2Occupied;
	tyP0950Simu.tyMcToAGV.tyBtnMag2Rdy.bValue				:= p_tyDTMagToAGV.bCI2Rdy;

	//Magazine #3 to AGV Communication
	tyP0950Simu.tyMcToAGV.tyBtnMag3Auto.bValue				:= p_tyDTMagToAGV.bCI3Auto;
	tyP0950Simu.tyMcToAGV.tyBtnMag3Empty.bValue				:= p_tyDTMagToAGV.bCI3MagazineFull;
	tyP0950Simu.tyMcToAGV.tyBtnMag3IncorrectModel.bValue	:= p_tyDTMagToAGV.bCI3IncorrectMagazineModel;
	tyP0950Simu.tyMcToAGV.tyBtnMag3Occupied.bValue			:= p_tyDTMagToAGV.bCI3Occupied;
	tyP0950Simu.tyMcToAGV.tyBtnMag3Rdy.bValue				:= p_tyDTMagToAGV.bCI3Rdy;

	//SOT
	tyP0950Simu.tySimu.tyBtnMagSOT1.tyBtnError.bValue	:= p_tyDO.bSOT1MagError;
	tyP0950Simu.tySimu.tyBtnMagSOT1.tyBtnRdy.bValue		:= p_tyDO.bSOT1MagReady;
	tyP0950Simu.tySimu.tyBtnMagSOT1.tyBtnAvail.bValue	:= p_tyDO.bSOT1MagAvailable;
	tyP0950Simu.tySimu.tyBtnMagSOT1.tyBtnSize.bValue	:= p_tyDO.bSOT1MagSizeLarge;

	tyP0950Simu.tySimu.tyBtnMagSOT2.tyBtnError.bValue	:= p_tyDO.bSOT2MagError;
	tyP0950Simu.tySimu.tyBtnMagSOT2.tyBtnRdy.bValue		:= p_tyDO.bSOT2MagReady;
	tyP0950Simu.tySimu.tyBtnMagSOT2.tyBtnAvail.bValue	:= p_tyDO.bSOT2MagAvailable;
	tyP0950Simu.tySimu.tyBtnMagSOT2.tyBtnSize.bValue	:= p_tyDO.bSOT2MagSizeLarge;

	tyP0950Simu.tySimu.tyBtnMagSOT3.tyBtnError.bValue	:= p_tyDO.bSOT3MagError;
	tyP0950Simu.tySimu.tyBtnMagSOT3.tyBtnRdy.bValue		:= p_tyDO.bSOT3MagReady;
	tyP0950Simu.tySimu.tyBtnMagSOT3.tyBtnAvail.bValue	:= p_tyDO.bSOT3MagAvailable;
	tyP0950Simu.tySimu.tyBtnMagSOT3.tyBtnSize.bValue	:= p_tyDO.bSOT3MagSizeLarge;

	//SOT1
	IF tyP0950Simu.tySimu.tyBtnSOT1.tyBtnInPos.bRtCompl THEN
		IF tyP0950Simu.tySimu.tyBtnSOT1.tyBtnInPos.bValue THEN
			tySOTSimulateSig1.tyBtnInPos := TRUE;
			tyP0950Simu.tySimu.tyBtnSOT1.tyBtnInPos.bRtCompl := FALSE;
		ELSE
			tySOTSimulateSig1.tyBtnInPos:= FALSE;
			tyP0950Simu.tySimu.tyBtnSOT1.tyBtnInPos.bRtCompl:= FALSE;
		END_IF
	END_IF

	IF tyP0950Simu.tySimu.tyBtnSOT1.tyBtnRdy.bRtCompl THEN
		IF tyP0950Simu.tySimu.tyBtnSOT1.tyBtnRdy.bValue THEN
			tySOTSimulateSig1.tyBtnRdy := TRUE;
			tyP0950Simu.tySimu.tyBtnSOT1.tyBtnRdy.bRtCompl := FALSE;
		ELSE
			tySOTSimulateSig1.tyBtnRdy := FALSE;
			tyP0950Simu.tySimu.tyBtnSOT1.tyBtnRdy.bRtCompl:= FALSE;
		END_IF
	END_IF

	IF tyP0950Simu.tySimu.tyBtnSOT1.tyBtnAvail.bRtCompl THEN
		IF tyP0950Simu.tySimu.tyBtnSOT1.tyBtnAvail.bValue THEN
			tySOTSimulateSig1.tyBtnAvail := TRUE;
			tyP0950Simu.tySimu.tyBtnSOT1.tyBtnAvail.bRtCompl := FALSE;
		ELSE
			tySOTSimulateSig1.tyBtnAvail:= FALSE;
			tyP0950Simu.tySimu.tyBtnSOT1.tyBtnAvail.bRtCompl:= FALSE;
		END_IF
	END_IF

	IF tyP0950Simu.tySimu.tyBtnSOT1.tyBtnError.bRtCompl THEN
		IF tyP0950Simu.tySimu.tyBtnSOT1.tyBtnError.bValue THEN
			tySOTSimulateSig1.tyBtnError := TRUE;
			tyP0950Simu.tySimu.tyBtnSOT1.tyBtnError.bRtCompl := FALSE;
		ELSE
			tySOTSimulateSig1.tyBtnError:= FALSE;
			tyP0950Simu.tySimu.tyBtnSOT1.tyBtnError.bRtCompl:= FALSE;
		END_IF
	END_IF

	//SOT2
	IF tyP0950Simu.tySimu.tyBtnSOT2.tyBtnInPos.bRtCompl THEN
		IF tyP0950Simu.tySimu.tyBtnSOT2.tyBtnInPos.bValue THEN
			tySOTSimulateSig2.tyBtnInPos := TRUE;
			tyP0950Simu.tySimu.tyBtnSOT2.tyBtnInPos.bRtCompl := FALSE;
		ELSE
			tySOTSimulateSig2.tyBtnInPos:= FALSE;
			tyP0950Simu.tySimu.tyBtnSOT2.tyBtnInPos.bRtCompl:= FALSE;
		END_IF
	END_IF

	IF tyP0950Simu.tySimu.tyBtnSOT2.tyBtnRdy.bRtCompl THEN
		IF tyP0950Simu.tySimu.tyBtnSOT2.tyBtnRdy.bValue THEN
			tySOTSimulateSig2.tyBtnRdy := TRUE;
			tyP0950Simu.tySimu.tyBtnSOT2.tyBtnRdy.bRtCompl := FALSE;
		ELSE
			tySOTSimulateSig2.tyBtnRdy := FALSE;
			tyP0950Simu.tySimu.tyBtnSOT2.tyBtnRdy.bRtCompl:= FALSE;
		END_IF
	END_IF

	IF tyP0950Simu.tySimu.tyBtnSOT2.tyBtnAvail.bRtCompl THEN
		IF tyP0950Simu.tySimu.tyBtnSOT2.tyBtnAvail.bValue THEN
			tySOTSimulateSig2.tyBtnAvail := TRUE;
			tyP0950Simu.tySimu.tyBtnSOT2.tyBtnAvail.bRtCompl := FALSE;
		ELSE
			tySOTSimulateSig2.tyBtnAvail:= FALSE;
			tyP0950Simu.tySimu.tyBtnSOT2.tyBtnAvail.bRtCompl:= FALSE;
		END_IF
	END_IF

	IF tyP0950Simu.tySimu.tyBtnSOT2.tyBtnError.bRtCompl THEN
		IF tyP0950Simu.tySimu.tyBtnSOT2.tyBtnError.bValue THEN
			tySOTSimulateSig2.tyBtnError := TRUE;
			tyP0950Simu.tySimu.tyBtnSOT2.tyBtnError.bRtCompl := FALSE;
		ELSE
			tySOTSimulateSig2.tyBtnError:= FALSE;
			tyP0950Simu.tySimu.tyBtnSOT2.tyBtnError.bRtCompl:= FALSE;
		END_IF
	END_IF

	//SOT3
	IF tyP0950Simu.tySimu.tyBtnSOT3.tyBtnInPos.bRtCompl THEN
		IF tyP0950Simu.tySimu.tyBtnSOT3.tyBtnInPos.bValue THEN
			tySOTSimulateSig3.tyBtnInPos := TRUE;
			tyP0950Simu.tySimu.tyBtnSOT3.tyBtnInPos.bRtCompl := FALSE;
		ELSE
			tySOTSimulateSig3.tyBtnInPos:= FALSE;
			tyP0950Simu.tySimu.tyBtnSOT3.tyBtnInPos.bRtCompl:= FALSE;
		END_IF
	END_IF

	IF tyP0950Simu.tySimu.tyBtnSOT3.tyBtnRdy.bRtCompl THEN
		IF tyP0950Simu.tySimu.tyBtnSOT3.tyBtnRdy.bValue THEN
			tySOTSimulateSig3.tyBtnRdy := TRUE;
			tyP0950Simu.tySimu.tyBtnSOT3.tyBtnRdy.bRtCompl := FALSE;
		ELSE
			tySOTSimulateSig3.tyBtnRdy := FALSE;
			tyP0950Simu.tySimu.tyBtnSOT3.tyBtnRdy.bRtCompl:= FALSE;
		END_IF
	END_IF

	IF tyP0950Simu.tySimu.tyBtnSOT3.tyBtnAvail.bRtCompl THEN
		IF tyP0950Simu.tySimu.tyBtnSOT3.tyBtnAvail.bValue THEN
			tySOTSimulateSig3.tyBtnAvail := TRUE;
			tyP0950Simu.tySimu.tyBtnSOT3.tyBtnAvail.bRtCompl := FALSE;
		ELSE
			tySOTSimulateSig3.tyBtnAvail:= FALSE;
			tyP0950Simu.tySimu.tyBtnSOT3.tyBtnAvail.bRtCompl:= FALSE;
		END_IF
	END_IF

	IF tyP0950Simu.tySimu.tyBtnSOT3.tyBtnError.bRtCompl THEN
		IF tyP0950Simu.tySimu.tyBtnSOT3.tyBtnError.bValue THEN
			tySOTSimulateSig3.tyBtnError := TRUE;
			tyP0950Simu.tySimu.tyBtnSOT3.tyBtnError.bRtCompl := FALSE;
		ELSE
			tySOTSimulateSig3.tyBtnError:= FALSE;
			tyP0950Simu.tySimu.tyBtnSOT3.tyBtnError.bRtCompl:= FALSE;
		END_IF
	END_IF

	//OutShutter Sim
	bSimuMod := TRUE;// shutter sim
	IF tyP0950Simu.tySimu.tyBtnInShutterSim.bValue THEN
		IF fbShutterSimChgOver.Q OR tyP0950Simu.tySimu.tyBtnInShutterSim.bRtCompl THEN
			tyP0950Simu.tySimu.tyBtnInShutterSim.bRtCompl := FALSE;
			fbShutterSimChgOver (IN:= FALSE);
			IF p_tyDI.bOutShutterCloseRS AND(p_tyDI.bOutShutterCloseRS2 OR p_tyNtParamCurr.bProjOutletShut2Prep = FALSE) AND
				(p_tyDI.bOutShutterCloseRS3 OR p_tyNtParamCurr.bProjOutletShut3Prep = FALSE) AND p_tyDI.bInShutterCloseRS THEN
				eInShutterAct  := PneuActRet;
				eOutShutterAct := PneuActRet;
				eOutShutterAct2 := PneuActRet;
				eOutShutterAct3 := PneuActRet;
			ELSIF p_tyDI.bOutShutterOpenRS AND (p_tyDI.bOutShutterOpenRS2 OR p_tyNtParamCurr.bProjOutletShut2Prep = FALSE) AND
				(p_tyDI.bOutShutterOpenRS3 OR p_tyNtParamCurr.bProjOutletShut3Prep = FALSE)AND p_tyDI.bInShutterOpenRS THEN
				eInShutterAct  := PneuActExt;
				eOutShutterAct := PneuActExt;
				eOutShutterAct2 := PneuActExt;
				eOutShutterAct3 := PneuActExt;
			END_IF
		ELSIF fbShutterSimChgOver.ET = T#5s THEN

		END_IF

		IF p_eOutShutterStatus = Done AND (p_eOutShutterStatus2 = Done OR p_tyNtParamCurr.bProjOutletShut2Prep = FALSE) AND
			(p_eOutShutterStatus3 = Done OR p_tyNtParamCurr.bProjOutletShut3Prep = FALSE) AND p_eInShutterStatus = Done THEN
			eInShutterAct  := PneuActIdle;
			eOutShutterAct := PneuActIdle;
			eOutShutterAct2 := PneuActIdle;
			eOutShutterAct3 := PneuActIdle;
			fbShutterSimChgOver (IN:= TRUE);
		END_IF
		fbShutterSimChgOver;
	ELSE
		eInShutterAct  := PneuActIdle;
		eOutShutterAct := PneuActIdle;
		eOutShutterAct2 := PneuActIdle;
		eOutShutterAct3 := PneuActIdle;

	END_IF

	//Test trav
	IF tyP0950Simu.tySimu.tyBtnTestTrav.bValue THEN
		CASE usiTestTravStep OF
			0:
				eTravAct		:= TravActGoDPos;

				IF p_eTravStat = TravActGoDPos AND p_eTravStatus = Done THEN
					eTravAct	:= TravActIdle;
					usiTestTravStep := 1;
				END_IF
			1:

				eTravAct		:= TravActGoFPos;

				IF p_eTravStat = TravActGoFPos AND p_eTravStatus = Done THEN
					eTravAct	:= TravActIdle;
					usiTestTravStep := 0;
				END_IF
		END_CASE
		diMnlTravNomSpd		:= 1500000;
	ELSE
		eTravAct		:= TravActIdle;
		diMnlTravNomSpd		:= 0;
	END_IF

	//NT- speed
	IF tyP0950Simu.tySimu.tyBtnNtParaWr2.bValue AND usiSimuNtStep = 0 THEN
		eTravAct		:= TravActIdle;
		p_diNtParamTravAutoSpd 		:= tyP0950Simu.tySimu.tyNumTravSpd.diValue;
		p_diNtParamLifterAutoSpd	:= tyP0950Simu.tySimu.tyNumLifterSpd.diValue;
		eNtWr := 3;
		IF p_eNtParamStat = 3 AND p_eNtParamStatus = Done THEN
			tyP0950Simu.tySimu.tyBtnNtParaWr2.bValue := FALSE;
			eNtWr := 0;
		END_IF
	END_IF

	//NT -addr and jobno
	IF tyP0950Simu.tySimu.tyBtnNtParaWr.bValue THEN
		p_sNtParamJobNo 		:= tyP0950Simu.tySimu.tyStringJobNo.sValue;
		p_usiNtParamNtAddr 		:= DINT_TO_USINT( tyP0950Simu.tySimu.tyNumAddr.diValue);
		CASE usiSimuNtStep OF
			0:
				eNtWr := 3;
				IF p_eNtParamStat = 3 AND p_eNtParamStatus = Done THEN
					eNtWr := 0;
					usiSimuNtStep := 1;
				END_IF
			1:
				IF  p_eNtParamStatus = Idle THEN
					eNtWr := 5;
				END_IF
				IF p_eNtParamStat = 5 AND p_eNtParamStatus = Done THEN
					eNtWr := 0;
					usiSimuNtStep := 2;
				END_IF
			2:
				p_eAct := 1; //refresh page
				IF eUIInit = UIInitialDone THEN
					p_eAct := 0;
					usiSimuNtStep := 0;
					tyP0950Simu.tySimu.tyBtnNtParaWr.bValue := FALSE;
				END_IF
		END_CASE

	END_IF
	//Bypassfor calibration
	bBypassShutForCalib := tyP0950Simu.tySimu.tyBtnBypassShutforCalib.bValue;

END_ACTION
```

#### Act_OptP0950RstMnl.st
```iecst
ACTION Act_OptP0950RstMnl:

	IF eCurrPage <> UIP0950Simu THEN
		bSimuMod := FALSE;
		tyP0950Simu.tySimu.tyBtnInShutterSim.bValue := FALSE;

		bAGVSimulationOn := FALSE;
		tyP0950Simu.tyAGVToMc.tyBtnAGVSimulateOn.bValue := FALSE;

		bAGVSimulateOnline := FALSE;
		tyP0950Simu.tyAGVToMc.tyBtnAGVOnline.bValue := FALSE;

		tyAGVSimulateSig.bVEHAuto := FALSE;
		tyP0950Simu.tyAGVToMc.tyBtnAGVAuto.bValue := FALSE;

		tyAGVSimulateSig.bVEH1Occupied := FALSE;
		tyP0950Simu.tyAGVToMc.tyBtnAGV1Occupied.bValue := FALSE;

		tyAGVSimulateSig.bVEH2Occupied := FALSE;
		tyP0950Simu.tyAGVToMc.tyBtnAGV2Occupied.bValue := FALSE;

		tyAGVSimulateSig.bVEH3Occupied := FALSE;
		tyP0950Simu.tyAGVToMc.tyBtnAGV3Occupied.bValue := FALSE;

		tyAGVSimulateSig.bVEHInPos1 := FALSE;
		tyP0950Simu.tyAGVToMc.tyBtnAGVInPos1.bValue := FALSE;

		tyAGVSimulateSig.bVEHInPos2 := FALSE;
		tyP0950Simu.tyAGVToMc.tyBtnAGVInPos2.bValue := FALSE;

		tyAGVSimulateSig.bVEHInPos3 := FALSE;
		tyP0950Simu.tyAGVToMc.tyBtnAGVInPos3.bValue := FALSE;

		tyP0950Simu.tySimu.tyBtnNtParaWr.bValue := FALSE;
		tyP0950Simu.tySimu.tyBtnNtParaWr2.bValue := FALSE;
		tyP0950Simu.tySimu.tyBtnTestTrav.bValue := FALSE;
	END_IF

END_ACTION
```

#### Act_OptP0950DispBffrCycle.st
```iecst
ACTION 	Act_OptP0950DispBffrCycle:
	IF tyP0950Simu.tySimuBffrCycleTm.tyDrpDnMagSel.usiValueIdx = 0 THEN
		p_tyBufferDispCycleTmBffr ACCESS p_Simu2DispCyclTmBffr1;
		p_bLocalMagPresent ACCESS ADR(p_tyDI.bMagPresentSen1);
	ELSIF tyP0950Simu.tySimuBffrCycleTm.tyDrpDnMagSel.usiValueIdx = 1 THEN
		p_tyBufferDispCycleTmBffr ACCESS p_Simu2DispCyclTmBffr2;
		p_bLocalMagPresent ACCESS ADR(p_tyDI.bMagPresentSen2);
	ELSIF tyP0950Simu.tySimuBffrCycleTm.tyDrpDnMagSel.usiValueIdx = 2 THEN
		p_tyBufferDispCycleTmBffr ACCESS p_Simu2DispCyclTmBffr3;
		p_bLocalMagPresent ACCESS ADR(p_tyDI.bMagPresentSen3);
	END_IF

//	tyP0950Simu.tySimuBffrCycleTm.tyTableList.tyUISlider.iMaxValue	:= DINT_TO_INT(p_tyBufferDispCycleTmBffr.diDispIdxEnd) - (c_uiP0950TableSize - 1);

	//Call Table FB
	fbP0950Table1.sVisuNm				:= tyP0950Table1.sVisuNm;
	fbP0950Table1.udiWorkAreaStartX		:= 15;
	fbP0950Table1.udiWorkAreaEndX		:= 365;
	fbP0950Table1.udiWorkAreaStartY		:= 109;
	fbP0950Table1.udiWorkAreaEndY		:= 429;
	fbP0950Table1.udiMinXDist			:= 20;
	fbP0950Table1.udiMinYDist			:= 20;
	fbP0950Table1.uiSlideScale			:= c_uiP0950TableSize;
	fbP0950Table1.iTotalData			:= DINT_TO_INT(p_tyBufferDispCycleTmBffr.diDispIdxEnd);
	fbP0950Table1.iTotalRow				:= c_uiP0950TableSize;
	fbP0950Table1(uiSliderStatus 		:= tyP0950Simu.tySimuBffrCycleTm.tyTableList.tyUISlider.uiRtStat , a_tyUIHotspot := tyP0950Simu.tySimuBffrCycleTm.tyTableList.a_tyHotspot , uiTablePos := tyP0950Table1.uiTablePos , iSliderPos := tyP0950Simu.tySimuBffrCycleTm.tyTableList.tyUISlider.iValue);

	tyP0950Table1.uiSelectedRow	:= fbP0950Table1.uiSelectedRow;
	tyP0950Table1.bTableActive	:= fbP0950Table1.bTableActive;
	tyP0950Table1.bSliderActive	:= fbP0950Table1.bSliderActive;

	//Table Content
	IF p_bLocalMagPresent  THEN
		FOR i := 1 TO c_uiP0950TableSize DO
			tyP0950Simu.tySimuBffrCycleTm.tyTableList.a_tyStringDataCol0[i].sValue		:= p_tyBufferDispCycleTmBffr.a_tyDispBffrDat[tyP0950Table1.uiTablePos + i - 1].sSlttoSltIdx;
			tyP0950Simu.tySimuBffrCycleTm.tyTableList.a_tyStringDataCol1[i].sValue		:= p_tyBufferDispCycleTmBffr.a_tyDispBffrDat[tyP0950Table1.uiTablePos + i - 1].sCycleTm;
			tyP0950Simu.tySimuBffrCycleTm.tyTableList.a_tyStringDataCol1[i].usiColor	:= DWORD_TO_USINT(p_tyBufferDispCycleTmBffr.a_tyDispBffrDat[tyP0950Table1.uiTablePos + i - 1].dwColor);

		END_FOR
	ELSE
		FOR i := 1 TO c_uiP0950TableSize DO
			tyP0950Simu.tySimuBffrCycleTm.tyTableList.a_tyStringDataCol0[i].sValue		:= '';
			tyP0950Simu.tySimuBffrCycleTm.tyTableList.a_tyStringDataCol1[i].sValue		:= '';
			tyP0950Simu.tySimuBffrCycleTm.tyTableList.a_tyStringDataCol1[i].usiColor	:= 0;

		END_FOR
	END_IF

	tyP0950Simu.tySimuBffrCycleTm.tyTableList.tyUISlider.iMaxValue	:= DINT_TO_INT(p_tyBufferDispCycleTmBffr.diDispIdxEnd) - (c_uiP0950TableSize - 1);

END_ACTION
```

#### Act_EntP1000Disp.st
```iecst
ACTION Act_EntP1000Disp:

	//Access Address
	p_tyC0005Main ACCESS ADR(tyCommon.tyMain);

	p_tyC0007Notif ACCESS ADR(tyCommon.tyNotif);

	p_tyC0008MsgBox ACCESS ADR(tyP1000Lang.tyMsgBoxHide);

	p_tyC0009Info ACCESS ADR(tyCommon.tyInfo);

	p_tyP1000Lang ACCESS ADR(tyP1000Lang.tyLang);

	//Backup Param
	tyP1000Lang.tyLangBkUp	:= tyP1000Lang.tyLang;

	//Display

	tyP1000Lang.tyLang.tyBtnEnglish.uiRtStat.0  :=  NOT(p_tyNtParamCurr.bChinesePrep OR p_tyNtParamCurr.bGermanPrep);
	tyP1000Lang.tyLang.tyBtnChinese.uiRtStat.0 := NOT(p_tyNtParamCurr.bChinesePrep);
	tyP1000Lang.tyLang.tyBtnGerman.uiRtStat.0  := NOT(p_tyNtParamCurr.bGermanPrep);

END_ACTION
```

#### Act_OptP1000SelectLang.st
```iecst
ACTION Act_OptP1000SelectLang:

	// Select English Language
	IF tyP1000Lang.tyLang.tyBtnEnglish.bRtCompl = TRUE THEN
		tyP1000Lang.tyLang.tyBtnEnglish.bRtCompl		:= FALSE;

		tyP1000Lang.tyLang.tyBtnEnglish.bValue			:= TRUE;
		tyP1000Lang.tyLang.tyBtnGerman.bValue			:= FALSE;
		tyP1000Lang.tyLang.tyBtnChinese.bValue			:= FALSE;

		tyP1000Lang.tyLang.tyBtnEnglish.bRtLk			:= TRUE;
		tyP1000Lang.tyLang.tyBtnGerman.bRtLk			:= FALSE;
		tyP1000Lang.tyLang.tyBtnChinese.bRtLk			:= FALSE;

		tyProperty.tyVisu.usiChgLang					:= 0;
		tyMcParamWr.usiLang								:= 0;

	// Select German Language
	ELSIF tyP1000Lang.tyLang.tyBtnGerman.bRtCompl = TRUE THEN
		tyP1000Lang.tyLang.tyBtnGerman.bRtCompl			:= FALSE;

		tyP1000Lang.tyLang.tyBtnEnglish.bValue			:= FALSE;
		tyP1000Lang.tyLang.tyBtnGerman.bValue			:= TRUE;
		tyP1000Lang.tyLang.tyBtnChinese.bValue			:= FALSE;

		tyP1000Lang.tyLang.tyBtnEnglish.bRtLk			:= FALSE;
		tyP1000Lang.tyLang.tyBtnGerman.bRtLk			:= TRUE;
		tyP1000Lang.tyLang.tyBtnChinese.bRtLk			:= FALSE;

		tyProperty.tyVisu.usiChgLang					:= 1;
		tyMcParamWr.usiLang								:= 1;

	// Select Chinese Language
	ELSIF tyP1000Lang.tyLang.tyBtnChinese.bRtCompl = TRUE THEN
		tyP1000Lang.tyLang.tyBtnChinese.bRtCompl		:= FALSE;

		tyP1000Lang.tyLang.tyBtnEnglish.bValue			:= FALSE;
		tyP1000Lang.tyLang.tyBtnGerman.bValue			:= FALSE;
		tyP1000Lang.tyLang.tyBtnChinese.bValue			:= TRUE;

		tyP1000Lang.tyLang.tyBtnEnglish.bRtLk			:= FALSE;
		tyP1000Lang.tyLang.tyBtnGerman.bRtLk			:= FALSE;
		tyP1000Lang.tyLang.tyBtnChinese.bRtLk			:= TRUE;

		tyProperty.tyVisu.usiChgLang					:= 2;
		tyMcParamWr.usiLang								:= 2;

	END_IF

END_ACTION
```

#### Act_OptP1000Keypad.st
```iecst
ACTION Act_OptP1000Keypad:

	IF fUIOutRtStatTPIsOpen(ADR(tyP1000Lang.tyLang.tyNumDay.uiRtStat)) = TRUE THEN
		tyProperty.tyKeypad.tyStringTitle.sKeypadTitle			:= tyP1000Lang.tyLang.tyNumDay.sKeypadTitle;

	ELSIF fUIOutRtStatTPIsOpen(ADR(tyP1000Lang.tyLang.tyNumMonth.uiRtStat)) = TRUE THEN
		tyProperty.tyKeypad.tyStringTitle.sKeypadTitle			:= tyP1000Lang.tyLang.tyNumMonth.sKeypadTitle;

	ELSIF fUIOutRtStatTPIsOpen(ADR(tyP1000Lang.tyLang.tyNumYear.uiRtStat)) = TRUE THEN
		tyProperty.tyKeypad.tyStringTitle.sKeypadTitle			:= tyP1000Lang.tyLang.tyNumYear.sKeypadTitle;

	ELSIF fUIOutRtStatTPIsOpen(ADR(tyP1000Lang.tyLang.tyNumSecond.uiRtStat)) = TRUE THEN
		tyProperty.tyKeypad.tyStringTitle.sKeypadTitle			:= tyP1000Lang.tyLang.tyNumSecond.sKeypadTitle;

	ELSIF fUIOutRtStatTPIsOpen(ADR(tyP1000Lang.tyLang.tyNumMinute.uiRtStat)) = TRUE THEN
		tyProperty.tyKeypad.tyStringTitle.sKeypadTitle			:= tyP1000Lang.tyLang.tyNumMinute.sKeypadTitle;

	ELSIF fUIOutRtStatTPIsOpen(ADR(tyP1000Lang.tyLang.tyNumHour.uiRtStat)) = TRUE THEN
		tyProperty.tyKeypad.tyStringTitle.sKeypadTitle			:= tyP1000Lang.tyLang.tyNumHour.sKeypadTitle;

	ELSE
		tyProperty.tyKeypad.tyStringTitle.sKeypadTitle			:= '';
	END_IF

END_ACTION
```

#### Act_EntP1020Disp.st
```iecst
ACTION Act_EntP1020Disp:

	//Access Address
	p_tyC0005Main ACCESS ADR(tyCommon.tyMain);

	p_tyC0007Notif ACCESS ADR(tyCommon.tyNotif);

	p_tyC0008MsgBox ACCESS ADR(tyP1020McSetNavi.tyMsgBoxHide);

	p_tyC0009Info ACCESS ADR(tyCommon.tyInfo);

	p_tyP1020McSetNavi ACCESS ADR(tyP1020McSetNavi.tyNavi);

	IF (p_tyNtParamCurr.bHermesSvyPrep AND p_tyMcParamCurr.bHermesSvyEn)
		OR p_tyNtParamCurr.bLFPrep OR p_tyNtParamCurr.bLCSLFPrep OR p_tyNtParamCurr.bLCSReqRcpPrep OR p_tyNtParamCurr.bLCSLiveDatPrep
		OR p_tyNtParamCurr.bLCSManageRcpPrep OR p_tyNtParamCurr.bLFUsrSetPrep OR p_tyNtParamCurr.bLFUsrSetPrep
		OR p_tyNtParamCurr.bUSWidthChkPrep OR p_tyNtParamCurr.bDSWidthChkPrep THEN

		fUIInRtStatOff(ADR(tyP1020McSetNavi.tyNavi.tyBtnVCommSet.uiRtStat));
	ELSE
		fUIInRtStatHide(ADR(tyP1020McSetNavi.tyNavi.tyBtnVCommSet.uiRtStat));
	END_IF

END_ACTION
```
